	//Команды текущего шага
	(*1*) cmd_KR12_Off := drm.cmd.0 := TRUE; //Закрытие крана 12, открытие крана 9
	(*1*) drm.error.0 := am.KR12.notOff OR am.KR9.notOn; //Кран 12 не закрылся, кран 9 не открылся

	//Условие перехода (5)→(6)
	//Кран 12 закрылся И кран 9 открылся
	IF (am.KR12.isOFF AND am.KR9.isON) AND drm.timeout THEN
		drm.cmd := drm.error := 0; drm.timer_pt := cycle; drm.inc := FALSE; drm.step := 6;
		cmd_KR12_Off := FALSE; //Закрытие крана 12, открытие крана 9
	END_IF;
6:	//Запись уставки таймера шага
	drm.step := 6;//Текущий шаг
	drm.timer_pt := cycle; //Таймер: один цикл вызова

	//Команды текущего шага
	(*1*) cmd_Kr6_Off := drm.cmd.0 := TRUE; //Кран 6 закрыть
	(*1*) drm.error.0 := am.Kr6.notOff; //Кран 6 не закрылся

	//Условие перехода (6)→(7)
	//Кран 6 закрыт
	IF (am.Kr6.isOFF) AND drm.timeout THEN
		drm.cmd := drm.error := 0; drm.timer_pt := cycle; drm.inc := FALSE; drm.step := 7;
		cmd_Kr6_Off := FALSE; //Кран 6 закрыть
	END_IF;
7:	//Запись уставки таймера шага
	drm.step := 7;//Текущий шаг
	drm.timer_pt := cycle; //Таймер: один цикл вызова

	//Команды текущего шага
	(*1*) cmd_Kr1_Off := drm.cmd.0 := TRUE; //Кран 1 закрыть
	(*1*) drm.error.0 := am.Kr1.notOff; //Кран 1 не закрылся

	(*2*) cmd_Kr2_Off := drm.cmd.1 := TRUE; //Кран 2 закрыть
	(*2*) drm.error.1 := am.Kr2.notOff; //Кран 2 не закрылся

	(*3*) cmd_Kr4_On := drm.cmd.2 := TRUE; //Кран 4 открыть
	(*3*) drm.error.2 := am.Kr4.notOn; //Кран 4 не открылся

	//Условие перехода (7)→(8)
	//Кран 1 закрыт И Кран 2 закрыт И Кран 4 открыт
	IF (am.Kr1.isOFF AND am.Kr2.isOFF AND am.Kr4.isON) AND drm.timeout THEN
		drm.cmd := drm.error := 0; drm.timer_pt := cycle; drm.inc := FALSE; drm.step := 8;
		cmd_Kr1_Off := FALSE; //Кран 1 закрыть
		cmd_Kr2_Off := FALSE; //Кран 2 закрыть
		cmd_Kr4_On := FALSE; //Кран 4 открыть
	END_IF;
8:	//Запись уставки таймера шага
	drm.step := 8;//Текущий шаг
	drm.timer_pt := cycle; //Таймер: один цикл вызова

	//Команды текущего шага
	(*1*) finish := drm.cmd.0 := TRUE; //Завершение

	//Условие перехода (8)→(0)
	//Логическая 1
	IF (TRUE) AND drm.timeout THEN
		drm.cmd := drm.error := 0; drm.timer_pt := cycle; drm.inc := FALSE; drm.step := -1;
		finish := FALSE; //Завершение
	END_IF;
END_CASE

//Принудительный выход из последовательности
IF break THEN
	drm.step := -1; drm.cmd := drm.error := 0; drm.timer_pt := cycle; drm.inc := FALSE;
	cmd_sound_On := FALSE; //Предпусковая сигнализация
	cmd_PNU_S_On := FALSE; //Пуск маслонасосов уплотнения и смазки
	cmd_sh_dPmg_On := FALSE; //Взвод защиты по перепаду "масло-газ"
	cmd_shPmN_On := FALSE; //Взвод защиты по маслосистеме нагнетателя
	cmd_filling := FALSE; //Запуск последовательности "Заполнение контура компрессора"
	cmd_KR12_On := FALSE; //Открытие крана 12, закрытие крана 9
	cmd_KR12_Off := FALSE; //Закрытие крана 12, открытие крана 9
	cmd_Kr6_Off := FALSE; //Кран 6 закрыть
	cmd_Kr1_Off := FALSE; //Кран 1 закрыть
	cmd_Kr2_Off := FALSE; //Кран 2 закрыть
	cmd_Kr4_On := FALSE; //Кран 4 открыть
	finish := FALSE; //Завершение
END_IF;

                  
END_FUNCTION_BLOCK

{region INFO}
(*
 Наименование последовательности: Переход К-М
 Автор: /Разработчик/ 08.08.2025 9:04:03
 Версия: v00.00.18
 Проект: KA107
*)
{endregion}
{attribute 'symbol' := 'none'}
FUNCTION_BLOCK PUBLIC T_K_M
VAR_INPUT
	cycle : REAL; //цикл вызова
END_VAR
VAR_OUTPUT
	cmd_Kr2_On : BOOL; //Кран 2 открыть
	cmd_Kr6_Off : BOOL; //Кран 6 закрыть
	finish : BOOL; //Завершение
	{attribute 'symbol' := 'read'}
	drm : Tdrm; //Интерфейсный функциональный блок
END_VAR
VAR
	start : BOOL; //Запуск последовательности
	break : BOOL; //Принудительный выход из последовательности
END_VAR

                    //Собираем переходы для визуализации
drm.transition.0 := start := mde.K_M; //Запуск последовательности (0→1): (Режим Переход К-М)
drm.transition.1 := am.Kr2.isON; //1→2: Кран 2 открыт
drm.transition.2 := am.Kr6.isOff; //2→3: Кран 6 закрыт
drm.transition.3 := TRUE; //3→0: Логическая 1
drm.transition.31 := break := alg.AO OR mde.M_K; //Принудительный выход из последовательности (N→0): Режимы аварийного останова ИЛИ Режим "Переход М-К"

//Вызываем экземпляр интерфейсного функционального блока
drm(cycle := cycle);

CASE drm.step OF
-1:	//Сброс команд с предыдущих шагов
	finish := FALSE;
	//Условие запуска последовательности
	//(Режим Переход К-М)
	IF start AND NOT break THEN drm.step := 1; END_IF;
1:	//Запись уставки таймера шага
	drm.step := 1;//Текущий шаг
	drm.timer_pt := cycle; //Таймер: один цикл вызова

	//Команды текущего шага
	(*1*) cmd_Kr2_On := drm.cmd.0 := TRUE; //Кран 2 открыть
	(*1*) drm.error.0 := am.Kr2.notOn; //Кран 2 не открылся

	//Условие перехода (1)→(2)
	//Кран 2 открыт
	IF (am.Kr2.isON) AND drm.timeout THEN
		drm.cmd := drm.error := 0; drm.timer_pt := cycle; drm.inc := FALSE; drm.step := 2;
		cmd_Kr2_On := FALSE; //Кран 2 открыть
	END_IF;
2:	//Запись уставки таймера шага
	drm.step := 2;//Текущий шаг
	drm.timer_pt := cycle; //Таймер: один цикл вызова

	//Команды текущего шага
	(*1*) cmd_Kr6_Off := drm.cmd.0 := TRUE; //Кран 6 закрыть
	(*1*) drm.error.0 := am.Kr6.notOff; //Кран 6 не закрылся

	//Условие перехода (2)→(3)
	//Кран 6 закрыт
	IF (am.Kr6.isOff) AND drm.timeout THEN
		drm.cmd := drm.error := 0; drm.timer_pt := cycle; drm.inc := FALSE; drm.step := 3;
		cmd_Kr6_Off := FALSE; //Кран 6 закрыть
	END_IF;
3:	//Запись уставки таймера шага
	drm.step := 3;//Текущий шаг
	drm.timer_pt := cycle; //Таймер: один цикл вызова

	//Команды текущего шага
	(*1*) finish := drm.cmd.0 := TRUE; //Завершение

	//Условие перехода (3)→(0)
	//Логическая 1
	IF (TRUE) AND drm.timeout THEN
		drm.cmd := drm.error := 0; drm.timer_pt := cycle; drm.inc := FALSE; drm.step := -1;
		finish := FALSE; //Завершение
	END_IF;
END_CASE

//Принудительный выход из последовательности
IF break THEN
	drm.step := -1; drm.cmd := drm.error := 0; drm.timer_pt := cycle; drm.inc := FALSE;
	cmd_Kr2_On := FALSE; //Кран 2 открыть
	cmd_Kr6_Off := FALSE; //Кран 6 закрыть
	finish := FALSE; //Завершение
END_IF;

                  
END_FUNCTION_BLOCK

{region INFO}
(*
 Наименование последовательности: Переход М-К
 Автор: /Разработчик/ 08.08.2025 9:04:03
 Версия: v00.00.18
 Проект: KA107
*)
{endregion}
{attribute 'symbol' := 'none'}
FUNCTION_BLOCK PUBLIC T_M_K
VAR_INPUT
	cycle : REAL; //цикл вызова
END_VAR
VAR_OUTPUT
	cmd_KR6_On : BOOL; //Кран 6 открыть
	cmd_Kr2_Off : BOOL; //Кран 2 закрыть
	finish : BOOL; //Завершение
	{attribute 'symbol' := 'read'}
	drm : Tdrm; //Интерфейсный функциональный блок
END_VAR
VAR
	start : BOOL; //Запуск последовательности
	break : BOOL; //Принудительный выход из последовательности
END_VAR

                    //Собираем переходы для визуализации
drm.transition.0 := start := mde.M_K OR NOss.cmd_M_K OR NObs.cmd_M_K; //Запуск последовательности (0→1): (Режим Переход М-К) ИЛИ (НОсс => Переход М-К) ИЛИ (НОбс => Переход М-К)
drm.transition.1 := am.Kr6.isON; //1→2: Кран 6 открыт
drm.transition.2 := am.Kr2.isOFF; //2→3: Кран 2 закрыт
drm.transition.3 := TRUE; //3→0: Логическая 1
drm.transition.31 := break := mde.AOss OR mde.AObs OR mde.K_M; //Принудительный выход из последовательности (N→0): Режим АОсс ИЛИ Режим АОбс ИЛИ Режим "Переход К-М"

//Вызываем экземпляр интерфейсного функционального блока
drm(cycle := cycle);

CASE drm.step OF
-1:	//Сброс команд с предыдущих шагов
	finish := FALSE;
	//Условие запуска последовательности
	//(Режим Переход М-К) ИЛИ (НОсс => Переход М-К) ИЛИ (НОбс => Переход М-К)
	IF start AND NOT break THEN drm.step := 1; END_IF;
1:	//Запись уставки таймера шага
	drm.step := 1;//Текущий шаг
	drm.timer_pt := cycle; //Таймер: один цикл вызова

	//Команды текущего шага
	(*1*) cmd_KR6_On := drm.cmd.0 := TRUE; //Кран 6 открыть
	(*1*) drm.error.0 := am.KR6.notOn; //Кран 6 не открылся

	//Условие перехода (1)→(2)
	//Кран 6 открыт
	IF (am.Kr6.isON) AND drm.timeout THEN
		drm.cmd := drm.error := 0; drm.timer_pt := cycle; drm.inc := FALSE; drm.step := 2;
		cmd_KR6_On := FALSE; //Кран 6 открыть
	END_IF;
2:	//Запись уставки таймера шага
	drm.step := 2;//Текущий шаг
	drm.timer_pt := cycle; //Таймер: один цикл вызова

	//Команды текущего шага
	(*1*) cmd_Kr2_Off := drm.cmd.0 := TRUE; //Кран 2 закрыть
	(*1*) drm.error.0 := am.Kr2.notOff; //Кран 2 не закрылся

	//Условие перехода (2)→(3)
	//Кран 2 закрыт
	IF (am.Kr2.isOFF) AND drm.timeout THEN
		drm.cmd := drm.error := 0; drm.timer_pt := cycle; drm.inc := FALSE; drm.step := 3;
		cmd_Kr2_Off := FALSE; //Кран 2 закрыть
	END_IF;
3:	//Запись уставки таймера шага
	drm.step := 3;//Текущий шаг
	drm.timer_pt := cycle; //Таймер: один цикл вызова

	//Команды текущего шага
	(*1*) finish := drm.cmd.0 := TRUE; //Завершение

	//Условие перехода (3)→(0)
	//Логическая 1
	IF (TRUE) AND drm.timeout THEN
		drm.cmd := drm.error := 0; drm.timer_pt := cycle; drm.inc := FALSE; drm.step := -1;
		finish := FALSE; //Завершение
	END_IF;
END_CASE

//Принудительный выход из последовательности
IF break THEN
	drm.step := -1; drm.cmd := drm.error := 0; drm.timer_pt := cycle; drm.inc := FALSE;
	cmd_KR6_On := FALSE; //Кран 6 открыть
	cmd_Kr2_Off := FALSE; //Кран 2 закрыть
	finish := FALSE; //Завершение
END_IF;

                  
END_FUNCTION_BLOCK

{region INFO}
(*
 Наименование последовательности: НОбс
 Автор: /Разработчик/ 08.08.2025 9:04:03
 Версия: v00.00.18
 Проект: KA107
*)
{endregion}
{attribute 'symbol' := 'none'}
FUNCTION_BLOCK PUBLIC T_NObs
VAR_INPUT
	cycle : REAL; //цикл вызова
END_VAR
VAR_OUTPUT
	cmd_M_K : BOOL; //Запуск последовательности "Переход М-К"
	sh_ms_off : BOOL; //Снятие защиты по маслосистеме ТК и СТ
	cooling : BOOL; //Охлаждение двигателя
	cmd_PNU_S_On : BOOL; //Включение маслонасосов смазки и уплотнения
	cmd_VNA_On : BOOL; //Включение Э/М ВНА
	cmd_KPV234_On : BOOL; //Открыть КПВ 2, 3, 4
	cmd_KR12_Off : BOOL; //Закрытие крана 12, открытие крана 9
	cmd_sh_TG_Off : BOOL; //Снятие защиты по ТГ
	cmd_SK_Off : BOOL; //СК закрыть
	check_Nst : BOOL; //Выбег нагнетателя
	cmd_Kr1_Off : BOOL; //Кран 1 закрыть
	cmd_Kr6_Off : BOOL; //Кран 6 закрыть
	cmd_Kr4_On : BOOL; //Кран 4 открыть
	check_Ntk : BOOL; //Выбег двигателя
	finish : BOOL; //Завершение
	{attribute 'symbol' := 'read'}
	drm : Tdrm; //Интерфейсный функциональный блок
END_VAR
VAR
	start : BOOL; //Запуск последовательности
	break : BOOL; //Принудительный выход из последовательности
END_VAR

                    //Собираем переходы для визуализации
drm.transition.0 := start := mde.NObs; //Запуск последовательности (0→1): Режим НОбс
drm.transition.1 := M_K.finish; //1→2: Последовательность "Переход М-К" завершена
drm.transition.2 := FuelReg.fReg.cooling; //2→3: Двигатель перешел на малый газ для охлаждения
drm.transition.3 := NOT FuelReg.fReg.cooling; //3→4: Охлаждение двигателя завершено
drm.transition.4 := am.KR9.ison AND am.KR12.isOff; //4→5: Подача топливного газа прекращена
drm.transition.5 := acpar.Nst.value < 100.0; //5→6: Nст < 100 об/мин
drm.transition.6 := am.Kr1.isOFF AND am.Kr6.isOFF AND am.Kr4.isON; //6→7: Кран 1 закрыт И Кран 6 закрыт И Кран 4 открыт
drm.transition.7 := acpar.Ntk.value < 100.0; //7→8: Nтк < 100 об/мин
drm.transition.8 := TRUE; //8→0: Логическая 1
drm.transition.31 := break := mde.AObs; //Принудительный выход из последовательности (N→0): Режим АОбс

//Вызываем экземпляр интерфейсного функционального блока
drm(cycle := cycle);

CASE drm.step OF
-1:	//Сброс команд с предыдущих шагов
	finish := FALSE;
	//Условие запуска последовательности
	//Режим НОбс
	IF start AND NOT break THEN drm.step := 1; END_IF;
1:	//Запись уставки таймера шага
	drm.step := 1;//Текущий шаг
	drm.timer_pt := cycle; //Таймер: один цикл вызова

	//Команды текущего шага
	(*1*) cmd_M_K := drm.cmd.0 := drm.step_time <= cycle; //Запуск последовательности "Переход М-К"

	//Условие перехода (1)→(2)
	//Последовательность "Переход М-К" завершена
	IF (M_K.finish) AND drm.timeout THEN
		drm.cmd := drm.error := 0; drm.timer_pt := cycle; drm.inc := FALSE; drm.step := 2;
		cmd_M_K := FALSE; //Запуск последовательности "Переход М-К"
	END_IF;
2:	//Запись уставки таймера шага
	drm.step := 2;//Текущий шаг
	drm.timer_pt := 10; //Таймер: 10 секунд

	//Команды текущего шага
	(*1*) sh_ms_off := drm.cmd.0 := TRUE; //Снятие защиты по маслосистеме ТК и СТ

	(*2*) alg.normalStopCom := drm.cmd.1 := TRUE; //Нормальный останов двигателя
	(*2*) drm.error.1 := NOT FuelReg.fReg.cooling; //Д не перешел на малый газ для охлаждения

	//Условие перехода (2)→(3)
	//Двигатель перешел на малый газ для охлаждения
	IF (FuelReg.fReg.cooling) AND drm.timeout THEN
		drm.cmd := drm.error := 0; drm.timer_pt := cycle; drm.inc := FALSE; drm.step := 3;
		sh_ms_off := FALSE; //Снятие защиты по маслосистеме ТК и СТ
	END_IF;
3:	//Запись уставки таймера шага
	drm.step := 3;//Текущий шаг
	drm.inc := TRUE; //Выставляем признак инкремента

	//Команды текущего шага
	(*1*) cooling := drm.cmd.0 := TRUE; //Охлаждение двигателя

	//Условие перехода (3)→(4)
	//Охлаждение двигателя завершено
	IF (NOT FuelReg.fReg.cooling) AND drm.timeout THEN
		drm.cmd := drm.error := 0; drm.timer_pt := cycle; drm.inc := FALSE; drm.step := 4;
		cooling := FALSE; //Охлаждение двигателя
	END_IF;
4:	//Запись уставки таймера шага
	drm.step := 4;//Текущий шаг
	drm.timer_pt := cycle; //Таймер: один цикл вызова

	//Команды текущего шага
	(*1*) alg.normalStopCom := FALSE; //Нормальный останов двигателя

	(*2*) cmd_PNU_S_On := drm.cmd.1 := TRUE; //Включение маслонасосов смазки и уплотнения

	(*3*) cmd_VNA_On := drm.cmd.2 := TRUE; //Включение Э/М ВНА

	(*4*) cmd_KPV234_On := drm.cmd.3 := TRUE; //Открыть КПВ 2, 3, 4
	(*4*) drm.error.3 := am.KPV2.notOn OR am.KPV3.notOn OR am.KPV4.notOn; //КПВ 2, 3, 4 не открылись

	(*5*) cmd_KR12_Off := drm.cmd.4 := TRUE; //Закрытие крана 12, открытие крана 9
	(*5*) drm.error.4 := am.KR12.notOff OR am.KR9.notOn; //Кран 12 не закрылся, кран 9 не открылся

	(*6*) cmd_sh_TG_Off := drm.cmd.5 := TRUE; //Снятие защиты по ТГ

	(*7*) cmd_SK_Off := drm.cmd.6 := TRUE; //СК закрыть

	//Условие перехода (4)→(5)
	//Подача топливного газа прекращена
	IF (am.KR9.ison AND am.KR12.isOff) AND drm.timeout THEN
		drm.cmd := drm.error := 0; drm.timer_pt := cycle; drm.inc := FALSE; drm.step := 5;
		cmd_PNU_S_On := FALSE; //Включение маслонасосов смазки и уплотнения
		cmd_KPV234_On := FALSE; //Открыть КПВ 2, 3, 4
		cmd_KR12_Off := FALSE; //Закрытие крана 12, открытие крана 9
		cmd_sh_TG_Off := FALSE; //Снятие защиты по ТГ
		cmd_SK_Off := FALSE; //СК закрыть
	END_IF;
5:	//Запись уставки таймера шага
	drm.step := 5;//Текущий шаг
	drm.timer_pt := cycle; //Таймер: один цикл вызова

	//Команды текущего шага
	(*1*) check_Nst := drm.cmd.0 := TRUE; //Выбег нагнетателя

	//Условие перехода (5)→(6)
	//Nст < 100 об/мин
	IF (acpar.Nst.value < 100.0) AND drm.timeout THEN
		drm.cmd := drm.error := 0; drm.timer_pt := cycle; drm.inc := FALSE; drm.step := 6;
		check_Nst := FALSE; //Выбег нагнетателя
	END_IF;
6:	//Запись уставки таймера шага
	drm.step := 6;//Текущий шаг
	drm.timer_pt := cycle; //Таймер: один цикл вызова

	//Команды текущего шага
	(*1*) cmd_Kr1_Off := drm.cmd.0 := TRUE; //Кран 1 закрыть
	(*1*) drm.error.0 := am.Kr1.notOff; //Кран 1 не закрылся

	(*2*) cmd_Kr6_Off := drm.cmd.1 := TRUE; //Кран 6 закрыть
	(*2*) drm.error.1 := am.Kr6.notOff; //Кран 6 не закрылся

	(*3*) cmd_Kr4_On := drm.cmd.2 := TRUE; //Кран 4 открыть
	(*3*) drm.error.2 := am.Kr4.notOn; //Кран 4 не открылся

	//Условие перехода (6)→(7)
	//Кран 1 закрыт И Кран 6 закрыт И Кран 4 открыт
	IF (am.Kr1.isOFF AND am.Kr6.isOFF AND am.Kr4.isON) AND drm.timeout THEN
		drm.cmd := drm.error := 0; drm.timer_pt := cycle; drm.inc := FALSE; drm.step := 7;
		cmd_Kr1_Off := FALSE; //Кран 1 закрыть
		cmd_Kr6_Off := FALSE; //Кран 6 закрыть
		cmd_Kr4_On := FALSE; //Кран 4 открыть
	END_IF;
7:	//Запись уставки таймера шага
	drm.step := 7;//Текущий шаг
	drm.timer_pt := cycle; //Таймер: один цикл вызова

	//Команды текущего шага
	(*1*) check_Ntk := drm.cmd.0 := TRUE; //Выбег двигателя

	//Условие перехода (7)→(8)
	//Nтк < 100 об/мин
	IF (acpar.Ntk.value < 100.0) AND drm.timeout THEN
		drm.cmd := drm.error := 0; drm.timer_pt := cycle; drm.inc := FALSE; drm.step := 8;
		check_Ntk := FALSE; //Выбег двигателя
	END_IF;
8:	//Запись уставки таймера шага
	drm.step := 8;//Текущий шаг
	drm.timer_pt := cycle; //Таймер: один цикл вызова

	//Команды текущего шага
	(*1*) cmd_VNA_On := FALSE; //Отключение Э/М ВНА

	(*2*) finish := drm.cmd.1 := drm.step_time <= cycle; //Завершение

	//Условие перехода (8)→(0)
	//Логическая 1
	IF (TRUE) AND drm.timeout THEN
		drm.cmd := drm.error := 0; drm.timer_pt := cycle; drm.inc := FALSE; drm.step := -1;
		finish := FALSE; //Завершение
	END_IF;
END_CASE

//Принудительный выход из последовательности
IF break THEN
	drm.step := -1; drm.cmd := drm.error := 0; drm.timer_pt := cycle; drm.inc := FALSE;
	cmd_M_K := FALSE; //Запуск последовательности "Переход М-К"
	sh_ms_off := FALSE; //Снятие защиты по маслосистеме ТК и СТ
	alg.normalStopCom := FALSE; //Нормальный останов двигателя
	cooling := FALSE; //Охлаждение двигателя
	cmd_PNU_S_On := FALSE; //Включение маслонасосов смазки и уплотнения
	cmd_VNA_On := FALSE; //Включение Э/М ВНА
	cmd_KPV234_On := FALSE; //Открыть КПВ 2, 3, 4
	cmd_KR12_Off := FALSE; //Закрытие крана 12, открытие крана 9
	cmd_sh_TG_Off := FALSE; //Снятие защиты по ТГ
	cmd_SK_Off := FALSE; //СК закрыть
	check_Nst := FALSE; //Выбег нагнетателя
	cmd_Kr1_Off := FALSE; //Кран 1 закрыть
	cmd_Kr6_Off := FALSE; //Кран 6 закрыть
	cmd_Kr4_On := FALSE; //Кран 4 открыть
	check_Ntk := FALSE; //Выбег двигателя
	finish := FALSE; //Завершение
END_IF;

                  
END_FUNCTION_BLOCK

{region INFO}
(*
 Наименование последовательности: НОсс
 Автор: /Разработчик/ 08.08.2025 9:04:03
 Версия: v00.00.18
 Проект: KA107
*)
{endregion}
{attribute 'symbol' := 'none'}
FUNCTION_BLOCK PUBLIC T_NOss
VAR_INPUT
	cycle : REAL; //цикл вызова
END_VAR
VAR_OUTPUT
	cmd_M_K : BOOL; //Запуск последовательности "Переход М-К"
	sh_ms_off : BOOL; //Снятие защиты по маслосистеме ТК и СТ
	cooling : BOOL; //Охлаждение двигателя
	cmd_PNU_S_On : BOOL; //Включение маслонасосов смазки и уплотнения
	cmd_VNA_On : BOOL; //Включение Э/М ВНА
	cmd_KPV234_On : BOOL; //Открыть КПВ 2, 3, 4
	cmd_KR12_Off : BOOL; //Закрытие крана 12, открытие крана 9
	cmd_sh_TG_Off : BOOL; //Снятие защиты по ТГ
	cmd_SK_Off : BOOL; //СК закрыть
	check_Nst : BOOL; //Выбег нагнетателя
	cmd_bleeding : BOOL; //Запуск последовательности "Стравливание контура компрессора"
	cmd_sh_dPmg_Off : BOOL; //Снятие защиты по перепаду "масло-газ"
	cmd_PNU_S_Off : BOOL; //Пуск таймера отключения ПНС, ПНУ
	check_Ntk : BOOL; //Выбег двигателя
	cmd_shPmN_Off : BOOL; //Снятие защиты по маслосистеме нагнетателя
	finish : BOOL; //Завершение
	{attribute 'symbol' := 'read'}
	drm : Tdrm; //Интерфейсный функциональный блок
END_VAR
VAR
	start : BOOL; //Запуск последовательности
	break : BOOL; //Принудительный выход из последовательности
END_VAR

                    //Собираем переходы для визуализации
drm.transition.0 := start := mde.NOss; //Запуск последовательности (0→1): Режим НОсс
drm.transition.1 := M_K.finish; //1→2: Последовательность "Переход М-К" завершена
drm.transition.2 := FuelReg.fReg.cooling; //2→3: Двигатель перешел на малый газ для охлаждения
drm.transition.3 := NOT FuelReg.fReg.cooling; //3→4: Охлаждение двигателя завершено
drm.transition.4 := am.KR9.ison AND am.KR12.isOff; //4→5: Подача топливного газа прекращена
drm.transition.5 := acpar.Nst.value < 100.0; //5→6: Nст < 100 об/мин
drm.transition.6 := bleeding.finish; //6→7: Подрежим "Стравливание контура компрессора" завершен
drm.transition.7 := acpar.Ntk.value < 100.0; //7→8: Nтк < 100 об/мин
drm.transition.8 := TRUE; //8→0: Логическая 1
drm.transition.31 := break := mde.AOss; //Принудительный выход из последовательности (N→0): Режим АОсс

//Вызываем экземпляр интерфейсного функционального блока
drm(cycle := cycle);

CASE drm.step OF
-1:	//Сброс команд с предыдущих шагов
	finish := FALSE;
	//Условие запуска последовательности
	//Режим НОсс
	IF start AND NOT break THEN drm.step := 1; END_IF;
1:	//Запись уставки таймера шага
	drm.step := 1;//Текущий шаг
	drm.timer_pt := cycle; //Таймер: один цикл вызова

	//Команды текущего шага
	(*1*) cmd_M_K := drm.cmd.0 := drm.step_time <= cycle; //Запуск последовательности "Переход М-К"

	//Условие перехода (1)→(2)
	//Последовательность "Переход М-К" завершена
	IF (M_K.finish) AND drm.timeout THEN
		drm.cmd := drm.error := 0; drm.timer_pt := cycle; drm.inc := FALSE; drm.step := 2;
		cmd_M_K := FALSE; //Запуск последовательности "Переход М-К"
	END_IF;
2:	//Запись уставки таймера шага
	drm.step := 2;//Текущий шаг
	drm.timer_pt := 10; //Таймер: 10 секунд

	//Команды текущего шага
	(*1*) sh_ms_off := drm.cmd.0 := TRUE; //Снятие защиты по маслосистеме ТК и СТ

	(*2*) alg.normalStopCom := drm.cmd.1 := TRUE; //Нормальный останов двигателя
	(*2*) drm.error.1 := NOT FuelReg.fReg.cooling; //Д не перешел на малый газ для охлаждения

	//Условие перехода (2)→(3)
	//Двигатель перешел на малый газ для охлаждения
	IF (FuelReg.fReg.cooling) AND drm.timeout THEN
		drm.cmd := drm.error := 0; drm.timer_pt := cycle; drm.inc := FALSE; drm.step := 3;
		sh_ms_off := FALSE; //Снятие защиты по маслосистеме ТК и СТ
	END_IF;
3:	//Запись уставки таймера шага
	drm.step := 3;//Текущий шаг
	drm.inc := TRUE; //Выставляем признак инкремента

	//Команды текущего шага
	(*1*) cooling := drm.cmd.0 := TRUE; //Охлаждение двигателя

	//Условие перехода (3)→(4)
	//Охлаждение двигателя завершено
	IF (NOT FuelReg.fReg.cooling) AND drm.timeout THEN
		drm.cmd := drm.error := 0; drm.timer_pt := cycle; drm.inc := FALSE; drm.step := 4;
		cooling := FALSE; //Охлаждение двигателя
	END_IF;
4:	//Запись уставки таймера шага
	drm.step := 4;//Текущий шаг
	drm.timer_pt := cycle; //Таймер: один цикл вызова

	//Команды текущего шага
	(*1*) alg.normalStopCom := FALSE; //Нормальный останов двигателя

	(*2*) cmd_PNU_S_On := drm.cmd.1 := TRUE; //Включение маслонасосов смазки и уплотнения

	(*3*) cmd_VNA_On := drm.cmd.2 := TRUE; //Включение Э/М ВНА

	(*4*) cmd_KPV234_On := drm.cmd.3 := TRUE; //Открыть КПВ 2, 3, 4
	(*4*) drm.error.3 := am.KPV2.notOn OR am.KPV3.notOn OR am.KPV4.notOn; //КПВ 2, 3, 4 не открылись

	(*5*) cmd_KR12_Off := drm.cmd.4 := TRUE; //Закрытие крана 12, открытие крана 9
	(*5*) drm.error.4 := am.KR12.notOff OR am.KR9.notOn; //Кран 12 не закрылся, кран 9 не открылся

	(*6*) cmd_sh_TG_Off := drm.cmd.5 := TRUE; //Снятие защиты по ТГ

	(*7*) cmd_SK_Off := drm.cmd.6 := TRUE; //СК закрыть

	//Условие перехода (4)→(5)
	//Подача топливного газа прекращена
	IF (am.KR9.ison AND am.KR12.isOff) AND drm.timeout THEN
		drm.cmd := drm.error := 0; drm.timer_pt := cycle; drm.inc := FALSE; drm.step := 5;
		cmd_PNU_S_On := FALSE; //Включение маслонасосов смазки и уплотнения
		cmd_KPV234_On := FALSE; //Открыть КПВ 2, 3, 4
		cmd_KR12_Off := FALSE; //Закрытие крана 12, открытие крана 9
		cmd_sh_TG_Off := FALSE; //Снятие защиты по ТГ
		cmd_SK_Off := FALSE; //СК закрыть
	END_IF;
5:	//Запись уставки таймера шага
	drm.step := 5;//Текущий шаг
	drm.timer_pt := cycle; //Таймер: один цикл вызова

	//Команды текущего шага
	(*1*) check_Nst := drm.cmd.0 := TRUE; //Выбег нагнетателя

	//Условие перехода (5)→(6)
	//Nст < 100 об/мин
	IF (acpar.Nst.value < 100.0) AND drm.timeout THEN
		drm.cmd := drm.error := 0; drm.timer_pt := cycle; drm.inc := FALSE; drm.step := 6;
		check_Nst := FALSE; //Выбег нагнетателя
	END_IF;
6:	//Запись уставки таймера шага
	drm.step := 6;//Текущий шаг
	drm.timer_pt := cycle; //Таймер: один цикл вызова

	//Команды текущего шага
	(*1*) cmd_bleeding := drm.cmd.0 := drm.step_time <= cycle; //Запуск последовательности "Стравливание контура компрессора"

	//Условие перехода (6)→(7)
	//Подрежим "Стравливание контура компрессора" завершен
	IF (bleeding.finish) AND drm.timeout THEN
		drm.cmd := drm.error := 0; drm.timer_pt := cycle; drm.inc := FALSE; drm.step := 7;
		cmd_bleeding := FALSE; //Запуск последовательности "Стравливание контура компрессора"
	END_IF;
7:	//Запись уставки таймера шага
	drm.step := 7;//Текущий шаг
	drm.timer_pt := 2; //Таймер: 2 секунд

	//Команды текущего шага
	(*1*) cmd_sh_dPmg_Off := drm.cmd.0 := TRUE; //Снятие защиты по перепаду "масло-газ"

	(*2*) cmd_PNU_S_Off := drm.cmd.1 := drm.step_time <= cycle; //Пуск таймера отключения ПНС, ПНУ

	(*3*) check_Ntk := drm.cmd.2 := TRUE; //Выбег двигателя

	//Условие перехода (7)→(8)
	//Nтк < 100 об/мин
	IF (acpar.Ntk.value < 100.0) AND drm.timeout THEN
		drm.cmd := drm.error := 0; drm.timer_pt := cycle; drm.inc := FALSE; drm.step := 8;
		cmd_sh_dPmg_Off := FALSE; //Снятие защиты по перепаду "масло-газ"
		cmd_PNU_S_Off := FALSE; //Пуск таймера отключения ПНС, ПНУ
		check_Ntk := FALSE; //Выбег двигателя
	END_IF;
8:	//Запись уставки таймера шага
	drm.step := 8;//Текущий шаг
	drm.timer_pt := cycle; //Таймер: один цикл вызова

	//Команды текущего шага
	(*1*) cmd_VNA_On := FALSE; //Отключение Э/М ВНА

	(*2*) cmd_shPmN_Off := drm.cmd.1 := TRUE; //Снятие защиты по маслосистеме нагнетателя

	(*3*) cmd_PNU_S_Off := drm.cmd.2 := drm.step_time <= cycle; //Пуск таймера отключения ПНС, ПНУ

	(*4*) finish := drm.cmd.3 := TRUE; //Завершение

	//Условие перехода (8)→(0)
	//Логическая 1
	IF (TRUE) AND drm.timeout THEN
		drm.cmd := drm.error := 0; drm.timer_pt := cycle; drm.inc := FALSE; drm.step := -1;
		cmd_shPmN_Off := FALSE; //Снятие защиты по маслосистеме нагнетателя
		cmd_PNU_S_Off := FALSE; //Пуск таймера отключения ПНС, ПНУ
		finish := FALSE; //Завершение
	END_IF;
END_CASE

//Принудительный выход из последовательности
IF break THEN
	drm.step := -1; drm.cmd := drm.error := 0; drm.timer_pt := cycle; drm.inc := FALSE;
	cmd_M_K := FALSE; //Запуск последовательности "Переход М-К"
	sh_ms_off := FALSE; //Снятие защиты по маслосистеме ТК и СТ
	alg.normalStopCom := FALSE; //Нормальный останов двигателя
	cooling := FALSE; //Охлаждение двигателя
	cmd_PNU_S_On := FALSE; //Включение маслонасосов смазки и уплотнения
	cmd_VNA_On := FALSE; //Включение Э/М ВНА
	cmd_KPV234_On := FALSE; //Открыть КПВ 2, 3, 4
	cmd_KR12_Off := FALSE; //Закрытие крана 12, открытие крана 9
	cmd_sh_TG_Off := FALSE; //Снятие защиты по ТГ
	cmd_SK_Off := FALSE; //СК закрыть
	check_Nst := FALSE; //Выбег нагнетателя
	cmd_bleeding := FALSE; //Запуск последовательности "Стравливание контура компрессора"
	cmd_sh_dPmg_Off := FALSE; //Снятие защиты по перепаду "масло-газ"
	cmd_PNU_S_Off := FALSE; //Пуск таймера отключения ПНС, ПНУ
	check_Ntk := FALSE; //Выбег двигателя
	cmd_shPmN_Off := FALSE; //Снятие защиты по маслосистеме нагнетателя
	cmd_PNU_S_Off := FALSE; //Пуск таймера отключения ПНС, ПНУ
	finish := FALSE; //Завершение
END_IF;

                  
END_FUNCTION_BLOCK

///
/// Назначение: 		Подготовка данных и вызхов обработчиков сигнализаций
/// Версия: 			00.00.00
/// Проект: 			КА107
FUNCTION Alarm_link : BOOL

                    //Деблокировка
unlock := tch.Unlock.value := btn.Unlock.out;

//Проверка защит
tch.CheckAlarm_on.value := btn.CheckAlarm_on.out OR tch.CheckAlarm_on.value AND NOT btn.CheckAlarm_off.out;
crs.common.CheckAlarm := alr.common.CheckAlarm := tch.CheckAlarm_on.value; 

// Подготовка данных для обработчиков сигнализаций	 
// Включение защиты по маслосистеме воздушного стартера
tmr.crsPmStarter_20.in 	:= am.Kr13.on;
alg.sh_Starter 			:= tmr.crsPmStarter_20.q;

// Защита по топливному газу
alg.sh_TG	:= ( Start_D.cmd_sh_TG_On OR alg.sh_TG ) AND NOT ( NOss.cmd_sh_TG_Off OR NObs.cmd_sh_TG_Off OR AOss.cmd_sh_TG_Off OR AObs.cmd_sh_TG_Off ) OR tch.GTDwork.value;

// Включение защиты по не розжигу (10 sec)
//tmr.crsNIgnition_10.IN	:= Start_D.cmd_sh_nIgnition AND NOT FuelReg.fReg.isFire;
alg.sh_nIgnition 		:= Start_D.cmd_sh_nIgnition AND NOT FuelReg.fReg.isFire; //tmr.crsNIgnition_10.Q;

// Включение защиты по не раскрутке (10 sec)
//tmr.crsNBoost_10.IN		:= ( Start_D.cmd_sh_nBoost OR tmr.crsNBoost_10.IN ) AND acpar.Ntk.value < 5600 AND am.SK.on;
alg.sh_nBoost			:= ( Start_D.cmd_sh_nBoost ) AND acpar.Ntk.value < 5600 AND am.SK.on; //tmr.crsNBoost_10.Q;

// Взвод защиты КПВ234 не закрыты
tmr.KPV234_wOpen.IN		:= ( Start_D.cmd_KPV234_Off OR tmr.KPV234_wOpen.IN ) AND NOT tmr.KPV234_wOpen.Q;
alg.KPV234_wOpen		:= ( tmr.KPV234_wOpen.Q OR alg.KPV234_wOpen ) AND NOT ( NOss.cmd_KPV234_On OR NObs.cmd_KPV234_On OR AOss.cmd_KPV234_On OR AObs.cmd_KPV234_On ) OR tch.GTDwork.value;

// Взвод защиты КПВ15 не закрыты
tmr.KPV15_wOpen.IN		:= ( acpar.NtkPrived.value > Ntk_KPV15Close OR tmr.KPV15_wOpen.IN ) AND NOT ( AOss.cmd_KPV15_On OR AObs.cmd_KPV15_On OR alg.normalStopCom );
alg.KPV15_wOpen			:= tmr.KPV15_wOpen.Q;

// Взвод защиты КПВ15 не открыты
tmr.KPV15_nOpen.IN		:= ( acpar.NtkPrived.value < Ntk_KPV15Open ) AND ( acpar.NtkPrived.value > Ntk_KPVClose );
alg.KPV15_nOpen			:= tmr.KPV15_nOpen.Q;

// Взвод защиты по давлению газа перед краном 13
alg.sh_Pg_inKR13		:= ( HP.cmd_VS_On OR Start_D.cmd_VS_On OR alg.sh_Pg_inKR13 ) AND NOT ( HP.cmd_VS_Off OR Start_D.cmd_VS_Off );

// Взвод защиты по давлению масла нагнетателя
alg.sh_PmN				:= ( KPK.cmd_shPmN_On OR HP.cmd_shPmN_On OR APK.cmd_shPmN_On OR alg.sh_PmN ) AND NOT ( HP.cmd_shPmN_Off OR NOss.cmd_shPmN_Off OR AOss.cmd_shPmN_Off OR Bleeding_full.cmd_shPmN_Off ) OR tch.GTDwork.value;

// Взвод защиты по давлению масла ТК и СТ
alg.sh_PmGTD			:= alg.KPV15_wOpen;

// Взвод защиты по давлению масла перед ДГ (САР)
alg.sh_SAR				:= alg.KPV234_wOpen;

// Взвод защиты по перепаду масло-газ
alg.sh_dPmg				:= ( KPK.cmd_sh_dPmg_On OR HP.cmd_sh_dPmg_On OR APK.cmd_sh_dPmg_On OR alg.sh_dPmg ) AND NOT ( HP.cmd_sh_dPmg_Off OR NOss.cmd_sh_dPmg_Off OR AOss.cmd_sh_dPmg_Off OR Bleeding_full.cmd_sh_dPmg_Off ) OR tch.Gas_N.value;

// Аварийный останов
alg.emergStopCom		:= AOss.emergStopCom OR AObs.emergStopCom;

// Вызов обработчиков сигнализаций
PPU_update(); // Предпусковые условия
ALR_update(); // Предупреждения
CRS_update(); // Аварии
                  
END_FUNCTION

FUNCTION ALG_D_link : BOOL

                    
subsystem.BD(
	goWork := FuelReg.fReg.start OR HP.cmd_HP_D,
	work := tch.GTDwork.value OR mde.HP AND acpar.Ntk.value > 500.0, 
	stop := acpar.Ntk.value < 100.0);
	
//Автоформируемый вызов последовательностей
bd_update(cycle := cycle_time_base);

ALG_D_AM_base();

// Сигнал "ГТД в работе"
tch.GTDwork.value 	:= FuelReg.fReg.started;
// Сигнал "Прогрев ГТД"
tch.GTDHeat.value	:= FuelReg.fReg.heating;
// Сигнал "Охлаждение двигателя"
tch.GTDcool.value	:= FuelReg.fReg.cooling;
// Сигнал "Пуск агрегата"
tch.GTDstart.value	:= FuelReg.fReg.start;

//engine.work8h(IN := tch.GTDwork.value);
//engine.work12h(IN := tch.GTDwork.value);

IF imitGPA.imit_on THEN D_imit(); END_IF;
                  
END_FUNCTION

///Chekmarev
FUNCTION D_imit : BOOL
VAR
	Tm		: REAL; //  
	///start		: BOOL;
	PmGood	: BOOL;
END_VAR
VAR CONSTANT
	/// максимальные обороты ТК на стартере
	Nstart_max: REAL := 2050;
	/// номинальные обороты ТК
	Ntk_norm: REAL := 8300;
	// нагрев масла нагревателем
	Ten		: REAL := 65;
	/// нагрев масла двигателем
	dTm_max: REAL := 26;
	tau_m: REAL := (300 * cycle_time_base);
	tau_mb: REAL := (5000 * cycle_time_base);
END_VAR

                    //start := am.Kr11.isON AND am.Kr10.isOFF AND am.Kr13.on;

// Раскрутка стартером
//IF am.SK.isOFF AND start THEN
//	aipar.Ntk_1.sim_value := aipar.Ntk_1.value + ( Nstart_max - aipar.Ntk_1.value ) / tau_start;
//END_IF

// Выбег двигателя
//IF am.SK.isOFF AND NOT start THEN
//	aipar.Ntk_1.sim_value := aipar.Ntk_1.value - aipar.Ntk_1.value / tau_stop;
//END_IF

//aipar.Ntk_2.sim_value := aipar.Ntk_1.value + ( 10 * BOOL_TO_BYTE (aipar.Ntk_1.value > 10.0 ));

// Температура масла
Tm	:= aipar.Tm_outAVOM.value;
aipar.Tm_MB.sim_value	:= aipar.Tm_MB.value + ( Tm - aipar.Tm_MB.value) / tau_mb;	// в маслобаке
aipar.Tm_outD.sim_value	:= aipar.Tm_outD.sim_value + (aipar.Tm_inD.value + dTm_max * ( acpar.Ntk.value / Ntk_norm) - aipar.Tm_outD.sim_value) / tau_m;
aipar.Tm_inD.sim_value	:= aipar.Tm_MB.value - 0.5;		// на входе в двигатель
Tm	:= aipar.Tm_outAVOM.value;
aipar.Tm_MBU.sim_value	:= aipar.Tm_MBU.value + ( Tm - aipar.Tm_MBU.value ) / ( tau_mb * 5 ); // маслобак уплотнений

// q = 160 кг в мин // расход
// Q = 8380000 дж в мин // передача теплоты в масло
// ~ 2000 дж/(кгС) // теплоемкость масла
// Итог:
// dt = ~26 градусов за мин

PmGood	:= acpar.Ntk.value > 5000;

dipar.Pm_N_An.sim_value	:= NOT ( am.PNS.isOn OR PmGood );
dipar.Pm_N_Pn.sim_value := NOT ( am.PNS.isOn OR acpar.Ntk.value > 6880 );
dipar.Pm_TK_An.sim_value := acpar.Ntk.value < 7700;
dipar.Pm_ST_An.sim_value := dipar.Pm_TK_An.value;

// БЗА Готовность 2
dipar.BZA_ready_2.sim_value	:= PmGood;

// Положение концевиков КПВ
dipar.KPV1_ON.sim_value	:= acpar.Ntk.value > Ntk_KPVClose AND acpar.Ntk.value < 7710;
dipar.KPV1_off.sim_value	:= NOT ( acpar.Ntk.value > Ntk_KPVClose AND acpar.Ntk.value < 7500 );

dipar.KPV2_ON.sim_value	:= am.KPV2.ON AND PmGood;
dipar.KPV2_off.sim_value	:= NOT dipar.KPV2_ON.value;

dipar.KPV3_ON.sim_value	:= am.KPV3.ON AND PmGood;
dipar.KPV3_off.sim_value	:= NOT dipar.KPV3_ON.value;

dipar.KPV4_ON.sim_value	:= am.KPV4.ON AND PmGood;
dipar.KPV4_off.sim_value	:= NOT dipar.KPV4_ON.value;

dipar.KPV5_ON.sim_value	:= dipar.KPV1_ON.value;
dipar.KPV5_off.sim_value	:= dipar.KPV1_off.value;
                  
END_FUNCTION

FUNCTION ALG_base : BOOL

                    //Предпусковые подрежимы
//Режимы
	ALG_Modes_link();

//Подсистемы
	ALG_EXT_Link();
	ALG_BTG_Link();
	ALG_MSD_link();
 	ALG_GO_link();
 	ALG_D_link();
 	ALG_BN_link();
	ALG_AVOM_Link();
	ALG_BPG_Link();
	ALG_VS_Link();
	ALG_VOU_Link();
	ALG_BU_Link();

//Подрежимы
	ALG_SMD_link();
	

	check_modes();	
//Общие ИМы
	ALG_AM();

//Имитация
	imit();

//Тестирование алгоритмов
//	test_function();
                  
END_FUNCTION

FUNCTION ALG_Modes_link : BOOL

                    //Вызов графа режимов	
mde_update();
mde_hmi.number := mde.number;
mde_hmi.status.0 := GVL_LIB.DU_prm_all;
mde_hmi.status.1 := GVL_LIB.sim_on_all;
mde_hmi.status.2 := alr.common.type_aggregated.1;
mde_hmi.status.3 := trs.common.type_aggregated.3 OR crs.common.aggregated;
mde_hmi.status.4 := lmt.common.type_aggregated.2 OR FuelReg.fReg.commonLimUp OR FuelReg.fReg.commonLimDn;
mde_hmi.status.5 := aipar.common.sim_aggregated OR aopar.common.sim_aggregated OR dipar.common.sim_aggregated OR dopar.common.sim_aggregated;
mde_hmi.status.6 := aipar.common.flt_aggregated;
mde_hmi.status.7 := aopar.common.flt_aggregated;
mde_hmi.status.8 := dipar.common.flt_aggregated;
mde_hmi.status.9 := dopar.common.flt_aggregated;

//Обобщенные сигналы
alg.stop := mde.AOss OR mde.AObs OR mde.NOss OR mde.NObs;
alg.reserve := mde.HR OR mde.GR;
alg.V_000 := alg.reserve OR mde.Repair;
alg.test := mde.HP OR mde.KPK;
alg.start := mde.APK;
alg.work := mde.K OR mde.M OR mde.K_M OR mde.M_K;
alg.AO := mde.AOss OR mde.AObs;
alg.NO := mde.NOss OR mde.NObs;
                  
END_FUNCTION

///
/// Назначение: 		Инициализация переменных
/// Автор: 			
/// Версия: 			00.00.01
FUNCTION fun_init : BOOL

                    
//Инициализация при запуске контроллера

btn.imit_ON.cmd := TRUE; //включение имитации

// Инициализация АВОМ
AVOM_Init();

// Запрет расчёта uccV на термопарах
aipar.Tg_inST_1.cfg.ucv_enabled := FALSE;
aipar.Tg_inST_2.cfg.ucv_enabled := FALSE;
aipar.Tg_inST_3.cfg.ucv_enabled := FALSE;
aipar.Tg_inST_4.cfg.ucv_enabled := FALSE;
aipar.Tg_inST_5.cfg.ucv_enabled := FALSE;
aipar.Tg_inST_6.cfg.ucv_enabled := FALSE;

// Инициализация FileManager
FilesNames.OperationTimePath := 'OpTime/';
FilesNames.OperationTimeFileExt := '.txt';
FilesNames.OperationTimeOut := 20000;	// Дпустимое время работы с файлами - 20 мс.
                  
END_FUNCTION

FUNCTION ALG_GO_AM : BOOL

                    
// Кран 1
am.Kr1.on 	:= Filling.cmd_Kr1_ON;
am.Kr1.off 	:= KPK.cmd_Kr1_Off OR NObs.cmd_Kr1_Off OR AObs.cmd_Kr1_Off OR Bleeding.cmd_Kr1_Off;
// Кран 1 смазка
dopar.Kr1m_ON.value	:= am.Kr1.offOut OR am.Kr1.onOut;

// Кран 2
//aspar.dP_Kr2.value := ABS(aipar.Pg_outN.value - aipar.Pg_aftKr2.value);
am.Kr2.on 	:= K_M.cmd_Kr2_ON;
am.Kr2.off	:= KPK.cmd_Kr2_Off OR M_K.cmd_Kr2_Off OR AObs.cmd_Kr2_Off OR Bleeding.cmd_Kr2_Off;
// Кран 2 смазка
dopar.Kr2m_ON.value	:= am.Kr2.offOut OR am.Kr2.onOut;

// Кран 4
am.Kr4.on 	:= Filling.cmd_Kr4_ON OR KPK.cmd_Kr4_ON OR NObs.cmd_Kr4_ON OR AObs.cmd_Kr4_ON;
am.Kr4.off 	:= Filling.cmd_Kr4_Off OR Bleeding.cmd_Kr4_Off OR AOss.cmd_Kr4_Off OR AObs.cmd_Kr4_Off;
// Кран 4 смазка
//dopar.Kr4m_ON.value	:= am.Kr4.offOut OR am.Kr4.onOut;

// Кран 5
am.Kr5.on 	:= Bleeding.cmd_Kr5_ON AND am.Kr6.isOFF;
am.Kr5.off 	:= Filling.cmd_Kr5_Off;
// Кран 5 смазка
//dopar.Kr5m_ON.value	:= am.Kr5.offOut OR am.Kr5.onOut;

// Кран 6
am.Kr6.on 	:= M_K.cmd_KR6_ON OR Filling.cmd_Kr6_ON OR s_tunpar.ASprot.emergOpenBypass;
am.Kr6.off 	:= K_M.cmd_Kr6_Off OR NObs.cmd_Kr6_Off OR Bleeding.cmd_Kr6_Off OR AObs.cmd_Kr6_Off OR KPK.cmd_Kr6_Off OR ( alg.KR6_off_after_emergOpenBypass.Qr AND mde.M );
// Кран 6 смазка
dopar.Kr6m_ON.value	:= am.Kr6.offOut OR am.Kr6.onOut;
                  
END_FUNCTION

///
/// Назначение: 		Управление крановой обвязкой
/// Автор: 			
/// Версия: 			00.00.01
FUNCTION ALG_GO_link : BOOL

                    
subsystem.GO(
	goWork := filling.start, 
	goStop := bleeding.start, 
	work := filling.finish, 
	stop := bleeding.finish);
//Автоформируемый вызов последовательностей
go_update(cycle := cycle_time_base);

//Исполнительные механизмы
ALG_GO_AM();

//Нет газа в контуре Компрессора
tch.nGas_N.value := aipar.Pg_inN.value < 0.05 AND aipar.Pg_outN.value < 0.05 AND dipar.Kr5_ON.value AND NOT dipar.Kr5_off.value;
//Газ в контуре Компрессора
tch.Gas_N.value := (aipar.Pg_inN.value > 0.2 OR aipar.Pg_outN.value > 0.2) AND dipar.Kr5_off.value AND NOT dipar.Kr5_ON.value OR aipar.Pg_inN.value > 0.2 AND aipar.Pg_outN.value > 0.2;

//Нет роста Рг на вх. К на 0,05 МПа в течении 10 сек
IF aipar.Pg_inN.value - Pg_inN_old < 0.05 THEN
	bn.delay_filling := bn.delay_filling + cycle_time_base;
	IF bn.delay_filling > 10.0 THEN bn.delay_filling := 0.0; alg.nIncPgN := TRUE; END_IF;
ELSE
	alg.nIncPgN := FALSE;
END_IF;
Pg_inN_old := aipar.Pg_inN.value;

// выделение заднего фронта (снятия) предпомпажной защиты
alg.KR6_off_after_emergOpenBypass.in := s_tunpar.ASprot.emergOpenBypass;

IF imitGPA.imit_on THEN GO_imit(); END_IF;
                  
END_FUNCTION

///Chekmarev
FUNCTION GO_imit : BOOL
VAR
	tau: REAL;
	p_in: REAL;
	kx: REAL;
END_VAR
VAR CONSTANT
	/// 30.6 кгс
	Pg_in: REAL := 3;
	Pg_out_max: REAL := 7;
	Nst_max: REAL := 8400;
END_VAR

                    
kx := (Pg_out_max - Pg_in) / Nst_max * BOOL_TO_INT( am.Kr6.isOFF );

//Давление газа в Н
IF NOT dipar.Kr5_off.value THEN 
	tau := 20.0; 
ELSIF dipar.Kr4_ON.value THEN 
	tau := 50.0; 
ELSIF (dipar.Kr1_ON.value OR dipar.Kr2_ON.value) THEN 
	tau := 10.0;  ELSE tau := 100.0; 
END_IF;

IF NOT dipar.Kr5_off.value THEN p_in := 0.0;
ELSIF dipar.Kr6_ON.value AND am.Kr6.isOFF THEN p_in := Pg_in;
ELSIF dipar.Kr4_ON.value OR dipar.Kr1_ON.value THEN p_in := Pg_in;
END_IF;

IF tau < 100.0 THEN 
	aipar.Pg_inN.sim_value := aipar.Pg_inN.sim_value + (p_in - aipar.Pg_inN.value) / (tau);
	aipar.Pg_outN.sim_value := aipar.Pg_inN.sim_value + acpar.Nst.value * kx;
END_IF; 

dipar.Pg_outKR1.sim_value := aipar.Pg_inN.value > 2.6;

//dipar.SK_OF.sim_value	:= am.SK.isOFF;
//dipar.SK_ON.sim_value	:= am.SK.isON;

//Т газа
aipar.Tg_inN.sim_value := aipar.Tg_inN.sim_value + (aipar.Ta_inK.value + aipar.Pg_inN.value * 4.2 - aipar.Tg_inN.sim_value)/(tau_det);
aipar.Tg_outN.sim_value := aipar.Tg_outN.sim_value + (aipar.Ta_inK.value + aipar.Pg_outN.value * 4.2 - aipar.Tg_outN.sim_value)/(tau_det);

IF aipar.Pg_inN.value < 0 THEN aipar.Pg_inN.sim_value := 0; END_IF;
IF aipar.Pg_outN.value < 0 THEN aipar.Pg_outN.sim_value := 0; END_IF;

                  
END_FUNCTION

FUNCTION ALG_BN_link : BOOL

                    
subsystem.BN(
	sys_type := 1,
	work := acpar.Nst.value > 20.0, 
	stop := acpar.Nst.value <= 20.0);
	
ALG_BN_base();
                  
END_FUNCTION

///
/// Назначение: 		Формирование выходных сигналов для сторожевого таймера
/// Автор: 			
/// Версия: 			00.00.01
FUNCTION ALG_PLC : BOOL
VAR
	cycle : REAL := GVL_LIB.cycle_time_fast;
END_VAR

                    
//Формирование меандра для реле БЭО
plc.BEO(tau := T#200MS, T := T#400MS, cycle := cycle);
dopar.BEO_w1.value := dopar.BEO_w2.value := plc.BEO.out;
                  
END_FUNCTION

///
/// Назначение: 		Вызов подрежимов
/// Автор: 			
/// Версия: 			00.00.01
FUNCTION ALG_SMD_link : BOOL

                    
//Функция обработки режимов и подрежимов с шагами
smd_update(cycle := cycle_time_base);
                  
END_FUNCTION

///
/// Назначение: 		Формирование выходных сигналов, не входящих ни в одну группу
/// Автор: 			
/// Версия: 			00.00.01
FUNCTION ALG_AM : BOOL

                    
dopar.Sound_ON.value := HP.cmd_sound_ON OR KPK.cmd_sound_ON OR APK.cmd_sound_ON;


                  
END_FUNCTION

FUNCTION ALG_D_AM_base : BOOL
VAR
	KPVOpen	: BOOL;
END_VAR

                    
//am.KPV1.on	:= ( AOss.cmd_KPV15_ON OR AObs.cmd_KPV15_ON OR am.KPV1.on ) AND NOT alg.V_000;
//am.KPV5.on	:= am.KPV1.on;

// Заглушка, т.к. КПВ1,5 управляются АУП-10
KPVOpen	:= ( acpar.NtkPrived.value > Ntk_KPVClose AND acpar.NtkPrived.value < Ntk_KPV15Open );
// КПВ 1
am.KPV1.on	:= KPVOpen;
// КПВ 2
am.KPV2.on	:= ( Start_D.cmd_KPV_On OR NOss.cmd_KPV234_ON OR NObs.cmd_KPV234_ON OR AOss.cmd_KPV234_ON OR AObs.cmd_KPV234_ON OR am.KPV2.on OR alg.V_000 ) AND NOT Start_D.cmd_KPV234_Off;
// КПВ 3
am.KPV3.on	:= am.KPV2.on;
// КПВ 4
am.KPV4.on	:= am.KPV2.on;
// КПВ 5
am.KPV5.on	:= KPVOpen;

// ВНА
am.VNA.on	:= Start_D.cmd_VNA_On OR NObs.cmd_VNA_On OR NOss.cmd_VNA_On OR AObs.cmd_VNA_On OR AOss.cmd_VNA_On;
// Обогрев ВНА
engine.VNAheat( par_value := aipar.Ta_inK.value, par_brk := aipar.Ta_inK.flt );
am.VNA_heat.on	:= ( engine.VNAheat.out OR dipar.Ace_alr.value ) AND NOT mde.Repair ;

// Агрегат зажигания
engine.AZ_off(IN := Start_D.cmd_AZ_ON);
am.AZ.on	:= engine.AZ_off.Q;
                  
END_FUNCTION

FUNCTION ALG_D_AM_fast : BOOL

                    // Стопорный клапан
//alg.SK_tr	:= (Start_D.cmd_SK_On OR alg.SK_tr) AND NOT (alg.AO OR alg.NO);
//am.SK.on	:= alg.SK_tr;

am.SK.on	:= (Start_D.cmd_SK_On OR am.SK.on) AND NOT (alg.AO OR NOss.cmd_SK_Off OR NObs.cmd_SK_Off);
                  
END_FUNCTION

{region INFO}
(*
 Назначение:   Используется для обработки аналоговых параметров, передаваемых с ВУ
 Автор:        /Разработчик/ 08.08.2025 8:32:24
 Конфигуратор: v00.01.00
 Проект:       KA107
*)
{endregion}
FUNCTION tunpar_update : BOOL
VAR_INPUT
END_VAR
VAR
END_VAR

                    tunpar.setNst(enable_direct_update := TRUE); //Задание Nst
tunpar.setNtk(enable_direct_update := TRUE); //Задание Ntk
tunpar.rateNstBtn(enable_direct_update := TRUE); //Шаг Nst для РЧВ
tunpar.rateNtkBtn(enable_direct_update := TRUE); //Шаг Ntk для РЧВ
tunpar.setTm(enable_direct_update := TRUE); //Задание температуры маслосистемы
tunpar.T1_avom(enable_direct_update := TRUE); //Т1 ПИД АВОМ
tunpar.T2_avom(enable_direct_update := TRUE); //Т2 ПИД АВОМ
tunpar.K_avom(enable_direct_update := TRUE); //К ПИД АВОМ
tunpar.DZ_avom(enable_direct_update := TRUE); //Зона нечувствительности ПИД АВОМ
tunpar.setTmMBDN(enable_direct_update := TRUE); //Температура в маслобаке смазки
tunpar.setTmMBN(enable_direct_update := TRUE); //Температура в маслобаке уплотнений
tunpar.countStart(enable_direct_update := TRUE); //Количество пусков
tunpar.countNO(enable_direct_update := TRUE); //Количество НО
tunpar.countAO(enable_direct_update := TRUE); //Количество АО
tunpar.generalOpTime(enable_direct_update := TRUE); //Наработка суммарная
tunpar.workOpTime(enable_direct_update := TRUE); //Наработка на режиме

                  
END_FUNCTION

FUNCTION tmr_update : BOOL

                    tmr.crsPmStarter_20();
//tmr.crsNIgnition_10();
//tmr.crsNBoost_10();
tmr.KPV15_nOpen();
tmr.KPV15_wOpen();
tmr.KPV234_wOpen();
tmr.PNU_S_Off();
tmr.PNU_S_pumpH();
                  
END_FUNCTION

{region INFO}
(*
 Назначение:   Ручной вызов обработчиков дискретных ИМов в fast цикле
 Автор:        /chekmarev/ 17.04.2025
 Проект:       KA107
*)
{endregion}
FUNCTION am_update_fast : BOOL

                    
//Стопорный клапан
//Тип: 1x2
am.SK(
	DU_prm := alg.V_000,
	onSigFlt := dipar.SK_ON.flt,
	onSig := dipar.SK_ON.value,
	onSig_sim_on := dipar.SK_ON.sim_on,
	onSig_sim_value := dipar.SK_ON.sim_value,
	offSigFlt	:= dipar.SK_off.flt,
	offSig		:= dipar.SK_off.value,
	offSig_sim_on:= dipar.SK_off.sim_on,
	offSig_sim_value := dipar.SK_off.sim_value,
	onFlt := dopar.SK_ON.flt);
dopar.SK_ON.value := am.SK.onOUT;
//--------------------------------------------------------------------------

//ДГ
//Тип: а
am.DG(
	PosSigFlt := aipar.DG_pos.flt,
	SetFlt := aopar.DG_set.flt,
	pos := aipar.DG_pos.value,
	pos_sim_on := aipar.DG_pos.sim_on,
	pos_sim_value := aipar.DG_pos.sim_value);
aopar.DG_set.value := am.DG.set_out;

 // Управление КПВ1, 5
dopar.KPV15_ON.value := ( am.KPV1.onOUT OR am.KPV5.onOut ) AND ( am.KPV1.DU AND am.KPV5.DU ) OR (( AOss.cmd_KPV15_ON OR AObs.cmd_KPV15_ON OR dopar.KPV15_ON.value ) AND NOT alg.V_000 );
// -----------------------------------
                  
END_FUNCTION

FUNCTION check_modes : BOOL

                    // Рп: Контроль ГР
PPU.Check_GR.value := (btn.GR.out OR NObs.finish OR HP.finish OR KPK.finish) OR PPU.Check_GR.value AND NOT (btn.HR.out OR btn.Repair.out OR btn.Start.out OR btn.Cancel.out OR alg.AO);

// Рп: Контроль ХР
PPU.Check_HR.value := (btn.HR.out OR btn.GR.out OR NObs.finish OR NOss.finish OR HP.finish OR KPK.finish) OR PPU.Check_HR.value AND NOT (btn.Repair.out OR btn.Start.out OR btn.Cancel.out OR alg.AO);

//Рп: Предпусковая готовность
check.btn := btn.HP.out OR btn.KPK.out OR btn.APK.out;
tch.PrepareStart.value := (check.btn OR tch.PrepareStart.value) AND NOT (btn.Start.out OR btn.Cancel.out OR mde.Repair);
   IF btn.HP.out THEN check.ready := ENUM_ReadyToStart.HP;
ELSIF btn.KPK.out THEN check.ready := ENUM_ReadyToStart.KPK;
ELSIF btn.APK.out THEN check.ready := ENUM_ReadyToStart.APK;
ELSIF NOT tch.PrepareStart.value THEN check.ready := ENUM_ReadyToStart.OFF;
END_IF;

//Рп: Сигналы готовности
tch.ReadyHP.value := ((check.ready = ENUM_ReadyToStart.HP AND tch.PrepareStart.value AND Check_SAU.finish) OR tch.ReadyHP.value) AND NOT (NOT (mde.GR OR mde.HR) OR btn.Cancel.out);
tch.ReadyKPK.value := ((check.ready = ENUM_ReadyToStart.KPK AND tch.PrepareStart.value AND Check_SAU.finish) OR tch.ReadyKPK.value) AND NOT (NOT (mde.GR OR mde.HR) OR btn.Cancel.out);
tch.ReadyAPK.value := ((check.ready = ENUM_ReadyToStart.APK AND tch.PrepareStart.value AND Check_SAU.finish) OR tch.ReadyAPK.value) AND NOT (NOT (mde.GR OR mde.HR) OR btn.Cancel.out);
check.ReadytoSF := tch.ReadyHP.value OR tch.ReadyKPK.value OR tch.ReadyAPK.value;


//Рп: Контроль САУ
//Проверка при подготовке к пуску или по кнопке при "Нет активных режимов" или каждые 12 часов, но не на пусковых режимах
check.tmr12H ( IN := NOT check.tmr12H.Q );
tch.Check_SAU.value := Check_SAU.drm.active;
check.tmrCancelPrm ( IN := Check_SAU.drm.active );
//Контроль виброаппаратуры двигателя (ИВ-Д-ПФ)
crs.Vs_D_Av.alg_check 	:= tch.Check_SAU.value;
crs.Vsst_HH.alg_check	:= tch.Check_SAU.value;
crs.Vstk_HH.alg_check	:= tch.Check_SAU.value;
crs.BZA_alr.alg_check	:= tch.Check_SAU.value;
dopar.Vibr_ctrl.value 	:= (Check_SAU.cmd_check_VibD OR dopar.Vibr_ctrl.value) AND NOT ( crs.Vs_D_Av.signalization AND crs.Vsst_HH.signalization AND crs.Vstk_HH.signalization OR btn.Cancel.out );
dopar.BZA_ctrl.value	:= (Check_SAU.cmd_check_BZA OR dopar.BZA_ctrl.value) AND NOT ( crs.BZA_alr.signalization OR btn.Cancel.out );
//tch.brk_vib_d.value := Check_SAU.cmd_check_VibD AND NOT (crs.VsPOD_OH.out AND crs.VsZOD_OH.out AND crs.VsD_Av.out);
//Разрешение старта
check.prm_start := (Check_SAU.finish AND check.ReadytoSF OR check.prm_start) AND NOT (btn.Start.out OR btn.Cancel.out OR mde.Repair);

//Имитация подрежима "Контроль САУ"
IF imitGPA.imit_on THEN check_imit(); END_IF;


                  
END_FUNCTION

FUNCTION check_imit : BOOL
VAR CONSTANT
	Ntk	: REAL := 8000;
END_VAR

                    check.tmrImit(IN := dopar.Vibr_ctrl.value OR dopar.BZA_ctrl.value);

dipar.Vs_D_Av.sim_value := check.tmrImit.Q;
dipar.BZA_alr.sim_value := check.tmrImit.Q;

aipar.Vstk.sim_value	:= TO_BYTE( check.tmrImit.Q ) * 92.0 + TO_REAL( SHR( PRG_base.result_time, 8) AND 2#00011111 ) * ( acpar.Ntk.value / Ntk );
aipar.Vsst.sim_value	:= aipar.Vstk.value;
                  
END_FUNCTION

FUNCTION_BLOCK TAcparHandler
VAR_INPUT
	/// в секундах 
	cycle: REAL;
END_VAR
VAR
	/// обработчики частот вращения 
	nTKfilter1: TMedianLagFilter;
	nTKfilter2: TMedianLagFilter;
	nSTfilter1: TMedianLagFilter;
	nSTfilter2: TMedianLagFilter;
	nTKcalc: TFreqRotorHandler;
	nSTcalc: TFreqRotorHandler;
END_VAR
VAR_TEMP
	// Среднее алгебраическое значение температуры
	TstAverage: REAL;
	// Количество исправных каналов
	TstCount: BYTE;	
END_VAR

                    (* фильтрация оборотов *)
(* нулевая постоянная времени фильтра тут корректна, при этом остается только медианный фильтр (чтобы убрать одиночные выбросы). 
При надобности можно увеличить tau, если нужен фильтр высокочастотной помехи (не отдельные "шилья", а "борода" на сигнале) *)
nTKfilter1( inVal:= aipar.Ntk_1.value, inBrk:= aipar.Ntk_1.flt, tau:= 0.3, cycle:= cycle ); 
nTKfilter2( inVal:= aipar.Ntk_2.value, inBrk:= aipar.Ntk_2.flt, tau:= 0.3, cycle:= cycle ); 
nSTfilter1( inVal:= aipar.Nst_1.value, inBrk:= aipar.Nst_1.flt, tau:= 0.3, cycle:= cycle ); 
nSTfilter2( inVal:= aipar.Nst_2.value, inBrk:= aipar.Nst_2.flt, tau:= 0.3, cycle:= cycle ); 

(* обработка двойных датчиков оборотов *)
nTKcalc.ch[1] 	:= nTKfilter1.outVal;
nTKcalc.ch[2]	:= nTKfilter2.outVal;
nTKcalc( disbal_Ch := 100.0, maxVal := aipar.Ntk_1.cfg.hilim, minVal := 100.0, ucvV := 500, flt_prm := acpar.Ntk.value > 500.0, deblock := btn.Unlock.out, out := acpar.Ntk );

nSTcalc.ch[1] 	:= nSTfilter1.outVal;
nSTcalc.ch[2]	:= nSTfilter2.outVal;
nSTcalc( disbal_Ch := 100.0, maxVal := aipar.Nst_1.cfg.hilim, minVal := 100.0, ucvV := 500, flt_prm := acpar.Nst.value > 500.0, deblock := btn.Unlock.out, out := acpar.Nst );

// обработка кольца термопар
{warning ' Убедиться, что в настройках модулей UCP1_A1_AI6 и UCP1_A1_AI7 выставлены диапазоны на каналах термопар (-50...+800) '}
// flt от модуля - обрыв или выход за пределы диапазона температур (-50...+800)
//TstCount := 0;
IF ( NOT aipar.Tg_inST_1.flt ) THEN
	TstAverage 	:= aipar.Tg_inST_1.value;
	TstCount 	:= 1;
END_IF
IF ( NOT aipar.Tg_inST_2.flt ) THEN
	TstAverage 	:= TstAverage + aipar.Tg_inST_2.value;
	TstCount	:= TstCount + 1;
END_IF
IF ( NOT aipar.Tg_inST_3.flt ) THEN
	TstAverage 	:= TstAverage + aipar.Tg_inST_3.value;
	TstCount	:= TstCount + 1;
END_IF
IF ( NOT aipar.Tg_inST_4.flt ) THEN
	TstAverage 	:= TstAverage + aipar.Tg_inST_4.value;
	TstCount	:= TstCount + 1;
END_IF
IF ( NOT aipar.Tg_inST_5.flt ) THEN
	TstAverage 	:= TstAverage + aipar.Tg_inST_5.value;
	TstCount	:= TstCount + 1;
END_IF
IF ( NOT aipar.Tg_inST_6.flt ) THEN
	TstAverage 	:= TstAverage + aipar.Tg_inST_6.value;
	TstCount	:= TstCount + 1;
END_IF

acpar.Tg_inST.flt 	:= TstCount = 0;
alg.TstInWork		:= TstCount;

IF TstCount > 0 THEN
	acpar.Tg_inST.in_value	:= TstAverage / TstCount;	
END_IF

(* все полученные данные выкладываются на входы acpar, acpar обновляются в своей автоматически сформированной функции *)
//acpar.Ntk.in_value := nVDcalc.value; acpar.Ntk.flt := nVDcalc.disbalanse;
//acpar.Nst.in_value := nSTcalc.value; acpar.Nst.flt := nSTcalc.disbalanse;
IF NOT aipar.Ta_inK.flt THEN acpar.NtkPrived.in_value := acpar.Ntk.value * SQRT( 288.15 / ( aipar.Ta_inK.value + 273.15 ) );
ELSE acpar.NtkPrived.in_value := acpar.Ntk.value;
END_IF;
acpar.Qtg_m3.in_value := FuelReg.fReg.fuel; 
                  
END_FUNCTION_BLOCK

FUNCTION_BLOCK TMedianLagFilter
VAR_INPUT
	inVal: REAL;
	inBrk: BOOL;
	tau: REAL;
	cycle: REAL;
END_VAR
VAR_OUTPUT
	outVal: REAL := 0;
END_VAR
VAR
	inArr: ARRAY[0..2] OF REAL;
	idx: INT := 0;
	cnt: INT;
	minVal: REAL := 1000000;
	maxVal: REAL := -1000000;
	sum: REAL;
END_VAR

                    IF inBrk THEN
	outVal := 0.0;
ELSE
  // заполнить входной массив, работает как кольцевой буфер
  inArr[ idx ] := inVal;
  idx := idx + 1;
  IF idx > 2 THEN idx := 0; END_IF;
  // сразу найти сумму - закладка под бОльщую размерность массива
  sum := 0.0;
  minVal := 1000000.0;
  maxVal := -1000000.0;
  FOR cnt := 0 TO 2 DO
	sum := sum + inArr[cnt];
    IF inArr[cnt] > maxVal THEN maxVal := inArr[cnt]; END_IF;  
    IF inArr[cnt] < minVal THEN minVal := inArr[cnt]; END_IF;  
  END_FOR
  // отбраковать минимум, максимум
  sum := sum - maxVal - minVal;
  // инерционное звено
  IF tau > cycle THEN
    outVal := outVal + ( cycle / tau ) * ( sum - outVal );	
  ELSE
	outVal := sum;   
  END_IF; 	
END_IF

                  
END_FUNCTION_BLOCK

FUNCTION FR_link : BOOL

                    // заполнение входных полей типа 
FuelReg.fReg.Nvd.value := acpar.Ntk.value; 
FuelReg.fReg.Nst.value:= acpar.Nst.value; 
FuelReg.fReg.Tg_outST.value:= acpar.Tg_inST.value; 
FuelReg.fReg.Pa_K.value:= aipar.Pa_out14.value; 
FuelReg.fReg.Ta_inD.value:= aipar.Ta_inK.value; 
FuelReg.fReg.Ttg_inValve.value := aipar.Ttg.value;
FuelReg.fReg.Ptg_inValve.value := aipar.Ptg_inTRK.value;
FuelReg.fReg.Nvd.flt := acpar.Ntk.flt; 
FuelReg.fReg.Nst.flt:= acpar.Nst.flt; 
FuelReg.fReg.Tg_outST.flt:= acpar.Tg_inST.flt; 
FuelReg.fReg.Pa_K.flt:= aipar.Pa_out14.flt; 
FuelReg.fReg.Ta_inD.flt:= aipar.Ta_inK.flt; 
FuelReg.fReg.Ttg_inValve.flt := aipar.Ttg.flt;
FuelReg.fReg.Ptg_inValve.flt := aipar.Ptg_inTRK.flt;

// обновление настроек
FuelRegTuns_update();

FuelReg.fReg(
	calcStep:= cycle_time_fast, 
    setValNvdExt:= tunpar.setNtk,  
	setValNstExt:= tunpar.setNst, 
	//startCom:= , // пишется в последовательностях
	checkCom := crs.Fire_flt.check,
    normalStopCom:= alg.normalStopCom, 
	emergStopCom:= alg.emergStopCom, 
	regNstOn:= bn.stabSTbtn, 
	fuel=>acpar.Qtg_m3.in_value, 
	setValve=>am.DG.set, 
	//start=> , // читается в последовательностях
	//heating=> , 
	//started=> , 
	//cooling=> , 
	//stoped=> , 
	//heatCountdown=> , 
	//coolCountdown=> , 
	//isFire=> 
     );
	 
FuelReg.fReg.update();	 


                  
END_FUNCTION

///
/// Назначение: 		Программный имитатор
/// Автор: 			
/// Версия: 			00.00.01
FUNCTION imit : BOOL
VAR CONSTANT
	tm: REAL := 15;
END_VAR

                    
//Инициализация
IF imitGPA.init (* OR testing.init *)THEN
	
	aipar.Tm_inD.sim_value	:= tm;
	aipar.Tm_MB.sim_value	:= tm;
	aipar.Tm_MBU.sim_value	:= tm;
	aipar.Tm_outAU.sim_value:= tm;
	aipar.Tm_outD.sim_value	:= tm;
	aipar.Tm_outAVOM.sim_value:= tm;
	
	aipar.Ta_inK.sim_value	:= tm;
	aipar.Tg_inST_1.sim_value := tm;
	aipar.Tg_inST_2.sim_value := tm + 2.3;
	aipar.Tg_inST_3.sim_value := tm - 1.2;
	aipar.Tg_inST_4.sim_value := tm;
	
	dipar.BZA_ready_1.sim_value		:= TRUE;
	dipar.Fuse_AO_UCP1.sim_value 	:= TRUE;
	dipar.Fuse_DO_UCP1.sim_value 	:= TRUE;
	dipar.Fuse_Air_UCP1.sim_value	:= TRUE;
	dipar.Fuse_DO_UE1.sim_value		:= TRUE;
	dipar.U_main.sim_value			:= TRUE;
	dipar.U_res.sim_value			:= TRUE;
	dipar.AG1.sim_value				:= TRUE;
	dipar.AG2.sim_value				:= TRUE;
	dipar.AG3.sim_value				:= TRUE;
	dipar.AG4.sim_value				:= TRUE;
	dipar.AG10.sim_value			:= TRUE;
	dipar.AG15.sim_value			:= TRUE;
	dipar.AG16.sim_value			:= TRUE;
	dipar.AG5.sim_value				:= TRUE;
	dipar.AG6.sim_value				:= TRUE;
	dipar.AG8.sim_value				:= TRUE;
	dipar.AG9.sim_value				:= TRUE;
	dipar.AG17.sim_value			:= TRUE;
	dipar.AG18.sim_value			:= TRUE;
	dipar.U_PRU.sim_value			:= TRUE;
	dipar.Utrk_main.sim_value		:= TRUE;
	dipar.U_AI.sim_value			:= TRUE;
	dipar.U_DI.sim_value			:= TRUE;
	dipar.U_BIZ.sim_value			:= TRUE;
	dipar.U_AM.sim_value			:= TRUE;
	dipar.Uvs_24.sim_value			:= TRUE;
	dipar.Uother_24.sim_value		:= TRUE;
	dipar.U_AM2.sim_value			:= TRUE;
	dipar.Utrk_res.sim_value		:= TRUE;
	dipar.Ubeo_main.sim_value		:= TRUE;
	dipar.Ubeo_res.sim_value		:= TRUE;
	dipar.AG11.sim_value			:= TRUE;
	dipar.AG12.sim_value			:= TRUE;
	dipar.U_KEAO.sim_value			:= TRUE;
	dipar.U_BEO.sim_value			:= TRUE;
	dipar.U_BZA.sim_value			:= TRUE;
	dipar.TRKready.sim_value		:= TRUE;
	
	dipar.EV1.sim_value				:= FALSE;
	dipar.EV2.sim_value				:= FALSE;
	dipar.EV3.sim_value				:= FALSE;
	dipar.EV4.sim_value				:= FALSE;
	dipar.Err_AUO1.sim_value		:= FALSE;
	
	dipar.Lm_MB_Pn.sim_value		:= FALSE;

	dipar.Lm_MBU_Pn.sim_value		:= FALSE;
	dipar.AO_PRU_2.sim_value		:= FALSE;
	dipar.Ace_alr.sim_value			:= FALSE;
	
	//Краны в положение останова
	am.Kr1.off 	:= TRUE;
	am.Kr2.off 	:= TRUE;
	am.Kr4.off 	:= TRUE;
	am.Kr5.on 	:= TRUE;	
	am.Kr6.off 	:= TRUE;
	am.Kr9.on 	:= TRUE;
	am.Kr10.on 	:= TRUE;
	am.Kr11.off := TRUE;
	am.Kr12.off := TRUE;
	am.KR13.off := TRUE;
	am.Kr15.off := TRUE;

	btn.Unlock.cmd := TRUE;
	imitGPA.init := FALSE;
END_IF;

IF imitGPA.imit_on THEN
	fun_ACS();
END_IF

//Включение имитации
imitGPA.imit_on := btn.imit_ON.out OR GVL_LIB.isTrainer OR imitGPA.imit_on AND NOT (btn.imit_OF.out);
gvl_lib.sim_on_all := imitGPA.imit_on;

//Переиницализация параметров начальными значениями при входе в имитацию
imitGPA.imit_start(CLK := imitGPA.imit_on);
imitGPA.init := imitGPA.imit_start.Q;
                  
END_FUNCTION

FUNCTION_BLOCK TImitEngineTuns
VAR_INPUT
	/// таблица открытия 
	openToGt: TLinear;
	GtToNvd: TLinear;
	GtToTst: TLinear;
	NvdToTauNvd: TLinear;
	NvdToTauTst: TLinear;
	NvdToTauPk: TLinear;
	NstToTauNst: TLinear;
	NvdToTst: TLinear;
	NvdToPk: TLinear;
	NvdToNst: TLinear;
	DUSdz: REAL;
	DUSrate: REAL;
	NvdStart: REAL;
END_VAR

                    
                  
END_FUNCTION_BLOCK

///2023-05-20
FUNCTION_BLOCK TEngineModel
VAR_INPUT
	/// температура атмосферного воздуха, ∞C
	Tatm: REAL;
	/// задание на ДГ, %
	setDG1: REAL;
	/// задание на ДГ, %
	setDG2: REAL;
	/// задание на ВНА, ∞
	setVNA: REAL;
	/// задание на  КПВ, ∞
	setKPV: REAL;
	/// призак работы стартера
	starter: BOOL;
	/// длЯ электростартера - работа на первой скорости
	starterSpeed1: BOOL;
	/// служебные сигналы, задающие конфигурацию ГТУ: наличие роторов среднего
	SDpresent: BOOL;
	/// и низкого давлениЯ газогенератора,
	NDpresent: BOOL;
	/// необходимость моделированиЯ давлениЯ за компрессором,
	PkPresent: BOOL;
	/// наличие дополнительного дозатора топлива,
	DUSaddPresent: BOOL;
	/// электростартер (по умолчанию - турбостартер)
	elStart: BOOL;
	cycle: REAL := cycle_time_fast;
	/// шаг интегрированиЯ в секундах 
	step: REAL;
	tuns: POINTER TO TImitEngineTuns;
END_VAR
VAR_OUTPUT
	/// расход топлива (кг/ч)
	Gfuel: REAL;
	/// положение ƒ√1, %
	posDG1: REAL;
	/// положение ƒ√1, %
	posDG2: REAL;
	/// положение ¬Ќј, ∞
	posVNA: REAL;
	/// положение  ѕ¬, ∞
	posKPV: REAL;
	/// частота вращения  Ќƒ, об/мин
	Nnd: REAL;
	/// среднего давлениЯ
	Nsd: REAL;
	/// частота вращения  ¬ƒ, об/мин
	Nvd: REAL;
	/// частота вращения —“, об/мин
	Nst: REAL;
	/// температура за “Ќƒ, ∞C
	Tt: REAL;
	/// температура за —“, ∞C
	Tst: REAL;
	/// давление за компрессором, ћѕа
	Pk: REAL;
	/// мощность двигателЯ в кВт
	power: REAL;
END_VAR
VAR
	/// зона нечувствительности привода ДУС (в %)
	DUS_DZ: REAL;
	/// скорость перемещениЯ привода ДУС (в %/с)
	DUS_RATE: REAL;
	NvdStart: REAL;
	/// расход топлива приведенный (кг/ч)
	Gt0: REAL;
	/// приведеннаЯ частота вращениЯ ротора ВД
	nvd0: REAL;
	/// частота вращениЯ ротора ВД, развиваемаЯ при раскрутке стартером
	NvdSetStarter: REAL;
	/// установившеесЯ значение частоты вращениЯ ротора ВД  
	nVDset: REAL;
	/// установившеесЯ значение температуры продуктов сгораниЯ перед СТ
	tSTset: REAL;
	tSTtoTT: REAL;
	/// количество шагов интегрированиЯ
	stepQuantity: DINT;
	/// счетчик шагов интегрированиЯ
	integCount: DINT;
	init: BOOL := FALSE;
	/// температура за ГГ на установившемся режиме
	Tt0: REAL;
END_VAR

                    IF NOT init THEN // инициализациЯ - производитсЯ считывание настроек, модель устанавливаетсЯ в нулевое начальное состоЯние
    DUS_DZ        := tuns^.DUSdz;
    DUS_RATE      := tuns^.DUSrate; 
    NvdStart := tuns^.NvdStart;
	tSTtoTT := 1.35; 
    Gt0  := 0.0;
    nvd0 := 0.1;
    NvdSetStarter := tuns^.NvdStart;
    nVDset := 0.1;
    tSTset := 0.0;
    posDG1 := 0.0;
    posDG2 := 0.0;
    nsd := 0.0;
    nnd := 0.0;
    nst := 0.0;
    init:= true;
    stepQuantity := REAL_TO_DINT(cycle/step + 0.5);
  ELSE // основнаЯ работа
    FOR integCount := 1 TO stepQuantity DO 
      // моделирование привода ДУСа (основного и дополнительного)
      // дозаторы топлива имеют шаговый электропривод с высоким быстродействием.
      IF nvd0 < 0.1 THEN nvd0 := 0.1; END_IF;
// Упрощаем имитацию ДУСа
//      DUSmdl(set := setDUSmain, dz := 0.25, cycle := step); 
      //YDUSmain := DUSmdl.out;
//      YDUSmain := setDUSmain;
      IF ABS( setDG1 - posDG1 ) > DUS_DZ THEN
        posDG1 := posDG1 + (step/( 0.3 * 100.0 / tuns^.DUSrate ) ) * (setDG1 - posDG1);		  
      END_IF;   
(* 
      IF setDG1 - posDG1 > DUS_DZ THEN
        posDG1 := posDG1 + step*DUS_RATE;
        IF posDG1 > setDG1 THEN posDG1 := setDG1; END_IF;
      ELSIF setDG1 - posDG1 < -DUS_DZ THEN
        posDG1 := posDG1 -step*DUS_RATE;
        IF posDG1 < setDG1 THEN posDG1 := setDG1; END_IF;
      END_IF;
      // длЯ двухзонных камер сгораниЯ: многозонность горениЯ не учитываетсЯ, а просто учитываетсЯ суммарный расход 
      //топлива через два дозатора
      IF DUSaddPresent THEN
        IF setDG2 - posDG2 > DUS_DZ THEN
          posDG2 := posDG2 + step*DUS_RATE;
          IF posDG2 > setDG2 THEN posDG2 := setDG2; END_IF;
        ELSIF setDG2 - posDG2 < -DUS_DZ THEN
          posDG2 := posDG2 -step*DUS_RATE;
          IF posDG2 < setDG2 THEN posDG2 := setDG2; END_IF;
        END_IF;
      END_IF;
      *)
	  tuns^.openToGt( arg := posDG1 + posDG2 );
      Gt0 := (tuns^.openToGt.out) * TO_INT(NOT dipar.SK_off.value);
      
      tuns^.GtToNvd(arg := Gt0 );
      tuns^.NvdToTauNvd(arg := Nvd);

      IF Gt0 < 0.0 THEN Gt0 := 0.0; END_IF;
  //    IF DUSaddPresent THEN Gt0 := Gt0 + tunings(tunName := tunConst.YDUSaddToGt, arg := YDUSadd); END_IF;
      // расход топлива
      // момент стартера
      IF starter THEN
        IF elStart THEN
          IF starterSpeed1 THEN NvdSetStarter := NvdStart/ 2.0;
          ELSE NvdSetStarter := NvdStart; END_IF;              
          // добавлено моделирование различной мощности электростартера на первой и второй скорости 
          IF NvdSetStarter > tuns^.GtToNvd.out THEN 
            nVDset := NvdSetStarter;
          ELSE nVDset := tuns^.GtToNvd.out;
          END_IF;       
        ELSE    
          nVDset := NvdStart + tuns^.GtToNvd.out;
        END_IF;  
      ELSE    
        nVDset := tuns^.GtToNvd.out;    
      END_IF;  
      // электростартер имеет почти постоЯнные обороты, поэтому обгоннаЯ муфта его
      // отключает. Турбостартер передает момент на вал всегда, когда включен
      // зубчатой муфтой и к нему подведен пусковой газ
      nvd0 := nvd0 + (step/(tuns^.NvdToTauNvd.out+0.001)) * (nVDset - nvd0);
      // частота вращениЯ ротора высокого давлениЯ (приведеннаЯ)
	  
      tuns^.GtToTst(arg := Gfuel);
      tuns^.NvdToTst(arg := Nvd);
      tuns^.NvdToTauTst(arg := Nvd);
	  
      tSTset := Tatm + tuns^.GtToTst.out - tuns^.NvdToTst.out;
	  IF tSTset < 0.0 THEN tSTset := 0.0; END_IF;
      Tst := Tst + (step/tuns^.NvdToTauTst.out) * (tSTset - Tst);
      // температура продуктов сгораниЯ вычислЯетсЯ в зависимости от частоты вращениЯ (-) и расхода топлива (+), учитываетсЯ
 
      Tt0 := tuns^.GtToTst.out - tuns^.NvdToTst.out;
      Tt  := Tt + (Tt0 - Tt) / tuns^.NvdToTauTst.out * cycle;

     // динамика
      nvd := nvd0 * SQRT((273.15 + Tatm)/288.15);
   (*   IF NDpresent THEN
        IF SDpresent THEN
          nsd := nsd + (step/(tunings(tunName := tunConst.nsdToTauSD, arg := nsd)+0.001))*
            (tunings(tunName := tunConst.nvdToNsd, arg := nvd) - nsd);
          nnd := nnd + (step/(tunings(tunName := tunConst.nndToTauND, arg := nnd)+0.001))*
            (tunings(tunName := tunConst.nsdToNnd, arg := nsd) - nsd);
        ELSE
          nsd := 0.0;
          nnd := nnd + (step/(tunings(tunName := tunConst.nsdToTauSD, arg := nnd)+0.001))*
            (tunings(tunName := tunConst.nvdToNsd, arg := nvd) - nnd); 
        END_IF;  
      END_IF;  
      // такаЯ хитраЯ логика свЯзана с терминологией: на двухвальных газогенераторах есть роторы ВД и НД, а на трехвальных - 
      // ВД, СД и НД. Поэтому, при наличии только флага НД игнорируетсЯ СД, а НД вычислЯетсЯ как СД.
	  *)	  	  
      IF PkPresent THEN
		tuns^.NvdToPk(arg := Nvd);
        tuns^.NvdToTauPk(arg := Nvd);
        Pk := Pk + (step/(tuns^.NvdToTauPk.out + 0.001)) * (tuns^.NvdToPk.out - Pk);
      END_IF;        
	  
	  
      (* пока не нужно, пригодится для генератора  
      power := tunings(tunName := tunConst.nvdToPower, arg := nvd0);
	  *)
      Gfuel := Gt0;
      // А здесь скорость СТ подсчитаем по упрощённой модели
 	  tuns^.NvdToNst(arg := Nvd);
      tuns^.NstToTauNst(arg := Nst);
      nst := nst + (step/(tuns^.NstToTauNst.out+0.001))*
                         (tuns^.NvdToNst.out - nst);
    END_FOR;
  END_IF; 	
	
	
                  
END_FUNCTION_BLOCK

FUNCTION_BLOCK TEdgeDetect
VAR_INPUT
	/// Вход импульсов
	in: BOOL;
END_VAR
VAR
	/// Передний край
	fe: BOOL;
	/// Задний край	
	re: BOOL;
	/// Предыдущее состояние входа
	oldin: BOOL;
	/// Промежуточное значение
	z: BOOL;
	/// Триггер переднего фронта 
	tf: BOOL;
	/// Триггер заднего фронта
	tr: BOOL;
END_VAR

                    z	:= in XOR oldIn;
fe	:= z AND in;
re	:= z AND oldin;
oldin := in;

tf	:= fe OR tf;	// tf и tr сбрасываем в акцессоре
tr	:= re OR tr;
                  

/// Выделение переднего фронта
PROPERTY Qf : BOOL
GET
                            Qf	:= tf;
tf	:= false;
                          
END_GET
SET
PRIVATE
                            
                          
END_SET
END_PROPERTY

/// Выделение заднего фронта
PROPERTY Qr : BOOL
GET
                            Qr	:= tr;
tr	:= false;
                          
END_GET
SET
PRIVATE
                            
                          
END_SET
END_PROPERTY
END_FUNCTION_BLOCK

FUNCTION ALG_BN_base : BOOL

                    // РЧВ
IF btn.turnDN.Qf THEN
	tunpar.setNst.set_value := tunpar.setNst.value - tunpar.rateNstBtn.value * TO_BYTE ( bn.stabSTbtn );
	tunpar.setNtk.set_value := tunpar.setNtk.value - tunpar.rateNtkBtn.value * TO_BYTE ( NOT bn.stabSTbtn );	
END_IF

IF btn.turnUP.Qf THEN
	tunpar.setNst.set_value := tunpar.setNst.value + tunpar.rateNstBtn.value * TO_BYTE ( bn.stabSTbtn );
	tunpar.setNtk.set_value := tunpar.setNtk.value + tunpar.rateNtkBtn.value * TO_BYTE ( NOT bn.stabSTbtn );
END_IF

IF NOT bn.stabSTbtn OR NOT tch.GTDwork.value THEN
	tunpar.setNst.value := acpar.Nst.value;
END_IF

IF bn.stabSTbtn OR NOT tch.GTDwork.value THEN
	tunpar.setNtk.value := acpar.Ntk.value;
END_IF

// Вытяжной вентилятор контейнера
am.VVN.on := dipar.Zagaz_OD_Pv.value;
bn.VVN_OFF( IN := NOT dipar.Zagaz_OD_Pv.value );
am.VVN.off:= bn.VVN_OFF.Q;
                  
END_FUNCTION

/// Маслоохладитель с дискретным включением вентиляторов
/// Вентиляторы включаются по наименьшей наработке
/// Выключаются - по наибольшей
/// Chekmarev
FUNCTION_BLOCK TAVOM
VAR_INPUT
	// разрешение работы АВОМ
	enable	: BOOL;
END_VAR
VAR_IN_OUT
	// Уставка температуры в маслосистеме
	Tm_SET	: Ttunpar;
	// Уставка Т1 для ПИД
	T1		: Ttunpar;
	// Уставка Т2 для ПИД
	T2		: Ttunpar;
	// Уставка K для ПИД
	K		: Ttunpar;
	// Уставка DZ для ПИД
	DZ		: Ttunpar;
	// Первый вентилятор маслоохладителя
	Vn1_AVOM: TAM_2x1;
	// Второй вентилятор маслоохладителя
	Vn2_AVOM: TAM_2x1;
	// Третий вентилятор маслоохладителя
	Vn3_AVOM: TAM_2x1;
	// Четвёртый вентилятор маслоохладителя
	Vn4_AVOM: TAM_2x1;	
END_VAR
VAR
	/// массив указателей на вентиляторы
	Vn_s: ARRAY[1..4] OF POINTER TO TAM_1x1;
	/// таймер отсчёта периода импульса
	tmrT: TON;
	/// Значение таймера на предыдущем цикле
	tmrT_Qold: BOOL;
	/// регулятор температуры масла
	TmReg: TPID;
	///	TmImp		: TP;		// инкремент / декремент счётчика
	///	target		: REAL;	
	_dz: REAL := 10;
	/// Флаг-указание на включение вентилятора из очереди
	_On: BOOL;
	/// Флаг-указание на отключение вентилятора из очереди
	_Off: BOOL;
END_VAR

                    
Vn_s[1]	:= ADR ( Vn1_AVOM );
Vn_s[2]	:= ADR ( Vn2_AVOM );
Vn_s[3]	:= ADR ( Vn3_AVOM );
Vn_s[4]	:= ADR ( Vn4_AVOM );
                  

METHOD PRIVATE PIDreg : BOOL
VAR_INPUT
	/// регулируемая температура
	temperature	: REAL;
END_VAR
VAR
	/// Ошибка регулирования	
	dTm: REAL;
END_VAR
                          // Регулирование с нуля
IF enable THEN
	TmReg.set_tun := FALSE;
	ELSE
		TmReg.set_tun	:= TRUE;
		TmReg.integ_tun	:= 0;
		TmReg.out_tun	:= 0;
END_IF

dTm := temperature - Tm_SET.value;

TmReg.setPID(_K := K.value, _T1 := T1.value, _T2 := T2.value, _DZ := DZ.value);
TmReg.singlePID(	err 	:= dTm,
					hiLimit	:= 100,
					loLimit	:= -100,
					hiRate	:= 10,
					loRate	:= 10,
					cycle	:= cycle_time_base,
					setDU	:= 0,
					DU		:= FALSE);
					
//target := TmReg.out;
                        
END_METHOD

/// Вентиляторы маслоохладителя
METHOD PRIVATE VnCntrl : BOOL
VAR
	index	: BYTE;
	min_	: BYTE := 1;
	max_	: BYTE := 1;
	on_1	: BOOL := TRUE;
	off_1	: BOOL := TRUE;
END_VAR
                          FOR index := 1 TO 4 DO
	Vn_s[index]^.on 	:= Vn_s[index]^.notOn AND Vn_s[index]^.flt;
	Vn_s[index]^.off 	:= FALSE;
END_FOR

IF On THEN
	FOR index := 1 TO 4 DO
	IF Vn_s[index]^.DU OR Vn_s[index]^.on THEN CONTINUE; END_IF
	IF Vn_s[index]^.isOFF THEN
		IF on_1 THEN
			min_ := index;
			on_1 := FALSE;
		END_IF
		IF Vn_s[index]^.OperationTime <= Vn_s[min_]^.OperationTime THEN
			min_ := index;
		END_IF
	END_IF
	END_FOR
	
	Vn_s[min_]^.off:= FALSE;
	Vn_s[min_]^.on := NOT Vn_s[min_]^.isON;
END_IF

IF Off THEN
	FOR index := 1 TO 4 DO
	IF Vn_s[index]^.DU OR Vn_s[index]^.off THEN CONTINUE; END_IF
	IF Vn_s[index]^.setOn THEN
		IF off_1 THEN
			max_ := index;
			off_1 := FALSE;
		END_IF
		IF ( Vn_s[index]^.OperationTime >= Vn_s[max_]^.OperationTime ) THEN
			max_ := index;
		END_IF
	END_IF
	END_FOR
	
	Vn_s[max_]^.on	:= FALSE;
	Vn_s[max_]^.off := Vn_s[max_]^.setOn; //NOT Vn_s[max_]^.isOFF OR Vn_s[max_]^.notOn;
END_IF
                        
END_METHOD

/// Chekmarev
METHOD update : BOOL
VAR_INPUT
	// регулируемая температура
	temperature	: REAL;
END_VAR
VAR
	// период следования импульсов
	T: TIME := TIME#1m0s0ms;
END_VAR
                          
PIDreg(temperature := temperature);

// Шаг импульса зависит от величины коррекции ошибки ПИД регулятором
// ( реализация ЧИМ )
T := TO_TIME (( 110 - ABS ( TmReg.out )) * 1000 );

tmrT ( in := NOT tmrT.Q, PT := T );

// Выделяем передний фронт импульса выхода таймера
IF (( tmrT.Q XOR tmrT_Qold ) AND tmrT.Q ) THEN
	IF ( 0 < tmreg.out - _DZ ) THEN
		_On 	:= TRUE;	// снимается в акцессоре
		_Off	:= FALSE;	// снимем на всякий случай
	END_IF
	
	IF ( 0 >= tmreg.out + _DZ ) THEN
		_On		:= FALSE;	// снимем на всякий случай
		_Off	:= TRUE;	// снимается в акцессоре
	END_IF
END_IF

tmrT_Qold := tmrT.Q;

IF NOT enable THEN
	_On	:= FALSE;
	_Off:= TRUE;
END_IF

VnCntrl();
                        
END_METHOD

/// Необходимо включить очередной вентилятор
PROPERTY On : BOOL
GET
PRIVATE
                            On		:= _On;
_On 	:= FALSE;
                          
END_GET
SET
PRIVATE
                            
                          
END_SET
END_PROPERTY

/// Необходимо выключить очередной вентилятор
PROPERTY Off : BOOL
GET
PRIVATE
                            Off		:= _Off;
_Off 	:= FALSE;
                          
END_GET
SET
PRIVATE
                            
                          
END_SET
END_PROPERTY
END_FUNCTION_BLOCK

PROGRAM PRG_PRU_Base
VAR_INPUT
	
	General: ARRAY[0..1] OF WORD := [4, 0];	/// номер агрегата [0] и режимх[1] 
	Holdings: ARRAY[0..16] OF REAL;
	Coils: ARRAY[0..13] OF BYTE;
	StatusReal: WORD;
END_VAR
VAR	
	Count: BYTE;	/// счётчик ошибок связи с ПРУ
	LinkPSU: BOOL;
	LinkPSUold: BOOL;
END_VAR

                    // Контроль связи с ПСУ
LinkPSU	:= Coils[13].1 XOR Coils[13].0;
IF LinkPSU THEN
	Count := Count + 1;
	ELSE
	Count := 0;
	PRU.Link := TRUE;
	LinkPSUold		:= NOT LinkPSUold;
END_IF

IF Count > 254 THEN 
	PRU.Link 	:= FALSE; 
	Count 		:= 1;
//	LinkPSUold		:= NOT LinkPSUold;
END_IF;

Coils[13].0	:= LinkPSUold;

// Кнопки
btn.AOss.cmd_PRU	:= Coils[0].0;//btn_AOss_Кнопка "АОсс"
btn.AObs.cmd_PRU	:= Coils[0].1;//btn_AObs_Кнопка "АОбс"
btn.NOss.cmd_PRU	:= Coils[0].2;//btn_NOss_Кнопка "НОсс"
btn.NObs.cmd_PRU	:= Coils[0].3;//btn_NObs_Кнопка "НОбс"
btn.turnUP.cmd_PRU	:= Coils[0].4;//btn_turnUP_Кнопка "Увеличить обороты"
btn.turnDN.cmd_PRU	:= Coils[0].5;//btn_turnDN_Кнопка "Уменьшить обороты"

//Coils[0].6;//btn_regNvd_Кнопка "Регулирование оборотов ВД"
//Coils[0].7;//btn_regNst_Кнопка "Регулирование оборотов СТ"
//Coils[1].0				:= btn.AOss_PRU;//prm_AOss_Разрешение кнопки "АОсс"
//Coils[1].1;//prm_AObs_Разрешение кнопки "АОбс"
//Coils[1].2;//prm_NOss_Разрешение кнопки "НОсс"
//Coils[1].3;//prm_NObs_Разрешение кнопки "НОбс"
Coils[1].4 := btn.turnUP.prm;//prm_turnUP_Разрешение кнопки "Увеличить обороты"
Coils[1].5 := btn.turnDN.prm;//prm_turnDN_Разрешение кнопки "Уменьшить обороты"
//Coils[1].6;//prm_regNvd_Разрешение кнопки "Регулирование оборотов ВД"
Coils[1].7 := btn.turnUP.prm OR btn.turnDN.prm;//prm_regNst_Разрешение кнопки "Регулирование оборотов СТ"

// ИМы
Coils[4].0		:= am.SK.isON;//NOT dipar_SK_OF_СК открыт
Coils[4].1		:= am.kr1.isON;//dipar_Kr1_ON_Кран КШ1 открыт
Coils[4].2		:= am.Kr1.isOFF;//dipar_Kr1_OF_Кран КШ1 закрыт
Coils[4].3		:= am.Kr2.isON;//dipar_Kr2_ON_Кран КШ2 открыт
Coils[4].4		:= am.Kr2.isOFF;//dipar_Kr2_OF_Кран КШ2 закрыт
Coils[4].5		:= am.Kr4.isON;//dipar_Kr4_ON_Кран КШ4 открыт
Coils[4].6		:= am.Kr4.isOFF;//dipar_Kr4_OF_Кран КШ4 закрыт
Coils[4].7		:= am.Kr5.isON;//dipar_Kr5_ON_Кран КШ5 открыт
Coils[5].0		:= am.Kr5.isOFF;//dipar_Kr5_OF_Кран КШ5 закрыт
Coils[5].1		:= am.Kr6.isON;//dipar_Kr6_ON_Кран КШ6 открыт
Coils[5].2		:= am.Kr6.isOFF;//dipar_Kr6_OF_Кран КШ6 закрыт
Coils[5].3		:= am.Kr9.isON;//dipar_Kr13_ON_Кран КШ13 открыт
Coils[5].4		:= am.Kr9.isOFF;//dipar_Kr13_OF_Кран КШ13 закрыт
Coils[5].5		:= am.Kr12.isON;//dipar_Kr14_ON_Кран КШ14 открыт
Coils[5].6		:= am.Kr12.isOFF;//dipar_Kr14_OF_Кран КШ14 закрыт

// Статусы подсистем
Coils[7].0	:= subsystem.EXT.nrml;	// status_EXT_nrml Внешние сигналы_норма
Coils[7].1	:= subsystem.EXT.alr;	// status_EXT_alr Внешние сигналы_предупрежденеие
Coils[7].2	:= subsystem.EXT.crs;	// status_EXT_crs Внешние сигналы_авария
Coils[7].3	:= subsystem.BD.nrml;	// status_BD_nrml Блок двигателя_норма
Coils[7].4	:= subsystem.BD.alr;	// status_BD_alr Блок двигателя_предупрежденеие
Coils[7].5	:= subsystem.BD.crs;	// status_BD_crs Блок двигателя_авария
Coils[7].6	:= subsystem.MSD.nrml;	// status_MSD_nrml Маслосистема двигателя_норма
Coils[7].7	:= subsystem.MSD.alr;	// status_MSD_alr Маслосистема двигателя_предупрежденеие
Coils[8].0	:= subsystem.MSD.crs;	// status_MSD_crs Маслосистема двигателя_авария
Coils[8].1	:= subsystem.BTG.nrml;	// status_BTG_nrml Блок топливного газа_норма
Coils[8].2	:= subsystem.BTG.alr;	// status_BTG_alr Блок топливного газа_предупрежденеие
Coils[8].3	:= subsystem.BTG.crs;	//status_BTG_crs Блок топливного газа_авария
Coils[8].4	:= subsystem.AVOM.nrml;//status_AVOMD_nrml АВОМД_норма
Coils[8].5	:= subsystem.AVOM.alr;//status_AVOMD_alr АВОМД_предупрежденеие
Coils[8].6	:= subsystem.AVOM.crs;//status_AVOMD_crs АВОМД_авария
Coils[8].7	:= subsystem.BN.nrml;//status_BN_nrml Блок нагнетателя_норма
Coils[9].0	:= subsystem.BN.alr;//status_BN_alr Блок нагнетателя_предупрежденеие
Coils[9].1	:= subsystem.BN.crs;//status_BN_crs Блок нагнетателя_авария
Coils[9].2	:= subsystem.GO.nrml;//status_GO_nrml Газовая обвязка_норма
Coils[9].3	:= subsystem.GO.alr;//status_GO_alr Газовая обвязка_предупрежденеие
Coils[9].4	:= subsystem.GO.crs;//status_GO_crs Газовая обвязка_авария
Coils[9].5	:= subsystem.VS.nrml;//status_VS_nrml Воздушный стартер_норма
Coils[9].6	:= subsystem.VS.alr;//status_VS_alr Воздушный стартер_предупрежденеие
Coils[9].7	:= subsystem.VS.crs;//status_VS_crs Воздушный стартер_авария
Coils[10].0	:= subsystem.BPG.nrml;//status_BPG_nrml Блок пускового газа_норма
Coils[10].1	:= subsystem.BPG.alr;//status_BPG_alr Блок пускового газа_предупрежденеие
Coils[10].2	:= subsystem.BPG.crs;//status_BPG_crs Блок пускового газа_авария
Coils[10].3	:= subsystem.POS.nrml;//status_POS_nrml ПОС ВОУ_норма
Coils[10].4	:= subsystem.POS.alr;//status_POS_alr ПОС ВОУ_предупрежденеие
Coils[10].5	:= subsystem.POS.crs;//status_POS_crs ПОС ВОУ_авария
Coils[10].6	:= subsystem.BU.nrml;//status_BU_nrml Блок автоматики_норма
Coils[10].7	:= subsystem.BU.alr;//status_BU_alr Блок автоматики_предупрежденеие
Coils[11].0	:= subsystem.BU.crs;//status_BU_crs Блок автоматики_авария


// Режим агрегата
General[1]			:= mde.number;

// Аналоги
//Holdings[1]		:= am.APK.pos; 				// aipar_APK_Pos_Положение клапана АПК1		// 2
//StatusReal.0	:= am.APK.flt;
//Holdings[2]		:= 0;			// aipar_reserve									// 4

//Holdings[3]		:= acpar.Ntk.value;		// acpar_evNnd_Расчётная Ntk				// 6
//StatusReal.2	:= acpar.Ntk.flt;

Holdings[4]		:= acpar.Ntk.value;		// acpar_evNvd_Расчётная Ntk				// 8
StatusReal.3	:= acpar.Nst.flt;

Holdings[5]		:= acpar.Nst.value;		// acpar_evNst_Расчётная Nст				// 10
StatusReal.4	:= acpar.Nst.flt;

Holdings[6]		:= aipar.Pg_inN.value;	// acpar_evPg_inN P газа на входе в компрессор		// 12
StatusReal.5	:= aipar.Pg_inN.flt;

Holdings[7]		:= aipar.Pg_outN.value;	// acpar_evPg_outN P газа на выходе из компрессора	// 14
StatusReal.6	:= aipar.Pg_outN.flt;

Holdings[8]		:= aipar.Tg_inN.value;	// acpar_evTg_inN T газа на входе в компрессор		// 16
StatusReal.7	:= aipar.Tg_inN.flt;

Holdings[9]		:= aipar.Tg_outN.value;	// acpar_evTg_outN T газа на выходе из компрессора	// 18
StatusReal.8	:= aipar.Tg_outN.flt;

//Holdings[10]	:= acpar.evdPg_conf.value;	// acpar_evdPg_conf_Расчётная dP газа на аннубар				// 20
//StatusReal.9	:= acpar.evdPg_conf.flt;

Holdings[11]	:= acpar.Tg_inST.value;	// acpar_evTg_outTND_Расчётная Т газа перед СТ					// 22
StatusReal.10	:= acpar.Tg_inST.flt;

//Holdings[12]	:= aipar.Ta_Angar.value;	// acpar_evTa_BN_Расчётная T воздуха в укрытии Компрессора		// 24
//StatusReal.11	:= aipar.Ta_Angar.flt;

Holdings[13]	:= aipar.Ta_inK.value;		// acpar_evTa_inBD_Расчётная T воздуха в блоке двигателя		// 26
StatusReal.12	:= aipar.Ta_inK.flt;

//Holdings[14]	:= s_aspar.surgeRes.value;	// acpar_Surge_Помпажный запас									// 28					
//StatusReal.13	:= s_aspar.surgeRes.flt;

IF aipar.Pg_inN.value > 0.0 THEN
	Holdings[15]	:= aipar.Pg_outN.value / aipar.Pg_inN.value;	// acpar_PR_Степень сжатия // 30
	ELSE 
		Holdings[15] := 0;
END_IF								
StatusReal.14	:= aipar.Pg_outN.flt OR aipar.Pg_inN.flt;		// s_aspar.evPR.flt;

Holdings[16]	:= aipar.Ptg_inTRK.value;	// aipar_Ptg_inD_Р топливного газа на вх. в Д	// 32
StatusReal.15	:= aipar.Ptg_inTRK.flt;

(*
Holdings[1]		:= Holdings[1] + 0.1; 				// aipar_APK_Pos_Положение клапана АПК1		// 2
//Holdings[2]		:= 0;			// aipar_reserve									// 4
Holdings[3]		:= Holdings[3] + 1; 			// acpar_evNnd_Расчётная Nвд							// 6
Holdings[4]		:= 3400;		// acpar_evNvd_Расчётная Nнд				// 8
Holdings[5]		:= 3001;		// acpar_evNst_Расчётная Nст				// 10
Holdings[6]		:= 6.6;	// acpar_evPg_inN_Расчётное P газа на входе в компрессор		// 12
Holdings[7]		:= 7.7;	// acpar_evPg_outN_Расчётное P газа на выходе из компрессора	// 14
Holdings[8]		:= 34.3;	// acpar_evTg_inN_Расчётная T газа на входе в компрессор		// 16
Holdings[9]		:= 87.9;	// acpar_evTg_outN_Расчётная T газа на выходе из компрессора	// 18
Holdings[10]	:= 20.01;	// acpar_evdPg_conf_Расчётная dP газа на аннубар				// 20
Holdings[11]	:= 470;	// acpar_evTg_outTND_Расчётная Т газа перед СТ					// 22
Holdings[12]	:= 22.12;	// acpar_evTa_BN_Расчётная T воздуха в укрытии Компрессора		// 24
Holdings[13]	:= 23.13;		// acpar_evTa_inBD_Расчётная T воздуха в блоке двигателя		// 26
Holdings[14]	:= 67.0;//	acpar. acpar_Surge_Помпажный запас									// 28					
Holdings[15]	:= 0.22;//acpar.PR; acpar_PR_Степень сжатия									// 30
Holdings[16]	:= 19.16;	// aipar_Ptg_inD_Р топливного газа на вх. в Д	// 32
*)
                  
END_PROGRAM

PROGRAM PRG_PRU_TimeSync
VAR
	///  Год, Месяц, День, час, минуты,секунды
	TimeAndDate: ARRAY[0..6] OF WORD;
	UnixTimems: DWORD;
	pres: UDINT;
	pDate: PsTime.SYSTIMEDATE;
END_VAR
VAR CONSTANT
	/// временная зона (в ПРУ Овен отсутствует)
	TimeZone: BYTE := 3;
END_VAR

                    // ---- Синхронизация времени
UnixTimems	:= PsTime.SysTimeRtcGet(pres);
PsTime.SysTimeRtcConvertUtcToDate(UnixTimems, pDate);

TimeAndDate[0]	:= pDate.wYear;				// Год
TimeAndDate[1]	:= pDate.wMonth;			// Месяц
TimeAndDate[2]	:= pDate.wDay;				// День
TimeAndDate[3]	:= pDate.wHour + TimeZone;	// Час
TimeAndDate[4]	:= pDate.wMinute;			// Минуты
TimeAndDate[5]	:= pDate.wSecond;			// Секунды

TimeAndDate[6]	:= 1;		// Признак готовности времени для синхронизации (признак снимается с ПРУ)

// ---- 
                  
END_PROGRAM

FUNCTION ALG_AVOM_Link : BOOL
VAR 
	temperature	: REAL;

END_VAR

                    subsystem.AVOM(
	goWork	:= am.Vn1_AVOM.on OR am.Vn2_AVOM.on OR am.Vn3_AVOM.on OR am.Vn4_AVOM.on,
	goStop	:= NOT ( am.Vn1_AVOM.on OR am.Vn2_AVOM.on OR am.Vn3_AVOM.on OR am.Vn4_AVOM.on ),
	work := am.Vn1_AVOM.isON OR am.Vn2_AVOM.isON OR am.Vn3_AVOM.isON OR am.Vn4_AVOM.isON,
	stop  := NOT ( am.Vn1_AVOM.isON OR am.Vn2_AVOM.isON OR am.Vn3_AVOM.isON OR am.Vn4_AVOM.isON )
);

//enable	:= mde.APK OR alg.work OR alg.NO OR am.PNU.isON OR am.PNS.isON;

avom.AVOM.enable	:= ( avom.AVOM.enable OR fuelreg.fReg.isFire ) AND NOT ( alg.V_000 AND am.PNS.isOFF AND am.PNU.isOFF ); 

temperature := MAX ( aipar.Tm_inD.value, aipar.Tm_outAU.value, aipar.Tm_outAVOM.value );
AVOM.AVOM.update( temperature := temperature );
IF imitGPA.imit_on THEN AVOM_imit(); END_IF;
                  
END_FUNCTION

FUNCTION AVOM_Imit : BOOL
VAR
	temp: REAL;
END_VAR

                    
temp := MAX (aipar.Tm_outD.value, aipar.Ta_inK.value);
aipar.Tm_outAVOM.sim_value	:= aipar.Tm_outAVOM.sim_value + ( temp - ( temp - aipar.Ta_inK.value) * ( TO_BYTE ( am.Vn1_AVOM.isON ) + TO_BYTE ( am.Vn2_AVOM.isON ) + TO_BYTE ( am.Vn3_AVOM.isON ) + TO_BYTE ( am.Vn4_AVOM.isON )) * 0.95 / 4 - aipar.Tm_outAVOM.sim_value ) / tau_Nto0;
aipar.Tm_outAU.sim_value 	:= aipar.Ta_inK.value;
                  
END_FUNCTION

FUNCTION AVOM_Init : BOOL

                    AVOM.AVOM ( Tm_SET		:= tunpar.setTm,
			T1			:= tunpar.T1_avom,
			T2			:= tunpar.T2_avom,
			K			:= tunpar.K_avom,
			DZ			:= tunpar.DZ_avom,
			Vn1_AVOM	:= am.Vn1_AVOM,
			Vn2_AVOM	:= am.Vn2_AVOM,
			Vn3_AVOM	:= am.Vn3_AVOM,
			Vn4_AVOM	:= am.Vn4_AVOM );
                  
END_FUNCTION

FUNCTION ALG_EXT_Link : BOOL

                    subsystem.EXT();
                  
END_FUNCTION

FUNCTION ALG_BTG_Link : BOOL

                    subsystem.BTG();

ALG_BTG_AM();

IF imitGPA.imit_on THEN BTG_imit(); END_IF;
                  
END_FUNCTION

FUNCTION ALG_MSD_link : BOOL

                    subsystem.MSD();

ALG_MSD_AM();

IF imitGPA.imit_on THEN MSD_imit(); END_IF;
                  
END_FUNCTION

FUNCTION MSD_Imit : BOOL
VAR CONSTANT
	dPmg_PNU: REAL := 0.7;
	dpmg_BN: REAL := 2.5;
	Nst_norm: REAL := 8500;
END_VAR

                    
aipar.dPmg.sim_value	:= (aipar.dPmg.value + (dPmg_PNU * BOOL_TO_BYTE( am.PNU.isOn ) + dpmg_BN * acpar.Nst.value / Nst_norm - aipar.dPmg.value) / tau_Po );
                  
END_FUNCTION

FUNCTION ALG_MSD_AM : BOOL

                    tmr.PNU_S_Off.IN 	:= ( NOss.cmd_PNU_S_Off OR AOss.cmd_PNU_S_Off OR Bleeding_full.cmd_PNU_S_Off OR tmr.PNU_S_Off.IN ) AND NOT ( tmr.PNU_S_Off.Q OR tch.Gas_N.value );
tmr.PNU_S_pumpH.IN	:= ( tch.GTDcool.value OR tch.GTDHeat.value ) AND dipar.Pm_N_Pn.value;

am.PNS.on	:= HP.cmd_PNU_S_On OR KPK.cmd_PNU_S_On OR APK.cmd_PNU_S_On OR NOss.cmd_PNU_S_On OR NObs.cmd_PNU_S_On OR AOss.cmd_PNU_S_On OR AObs.cmd_PNU_S_On OR ( mde.GR AND am.PNS.isOFF ) OR tmr.PNU_S_pumpH.IN;
am.PNS.off	:= (( HP.cmd_PNS_Off OR ( mde.HR OR mde.Repair ) AND am.PNS.isON AND tch.nGas_N.value ) AND NOT tmr.PNU_S_Off.IN ) OR Start_D.cmd_PNS_Off OR ( tmr.PNU_S_Off.Q AND tch.nGas_N.value ) OR (( tch.GTDcool.value OR tch.GTDHeat.value OR alg.work ) AND NOT tmr.PNU_S_pumpH.Q AND am.PNS.isON );

am.PNU.on	:= HP.cmd_PNU_S_On OR KPK.cmd_PNU_S_On OR APK.cmd_PNU_S_On OR NOss.cmd_PNU_S_On OR NObs.cmd_PNU_S_On OR AOss.cmd_PNU_S_On OR AObs.cmd_PNU_S_On OR ( mde.GR AND am.PNU.isOFF ) OR tmr.PNU_S_pumpH.IN;
am.PNU.off	:= (( HP.cmd_PNU_Off OR ( mde.HR OR mde.Repair ) AND am.PNU.isON AND tch.nGas_N.value ) AND NOT tmr.PNU_S_Off.IN ) OR Start_D.cmd_PNU_Off OR ( tmr.PNU_S_Off.Q AND tch.nGas_N.value ) OR (( tch.GTDcool.value OR tch.GTDHeat.value OR alg.work ) AND NOT tmr.PNU_S_pumpH.Q AND am.PNU.isON );

// Обогрев маслобака системы смазки
engine.ENBDN( par_value := aipar.Tm_MB.value, par_brk := aipar.Tm_MB.flt, setpoint_value := tunpar.setTmMBDN.value );
engine.ENBDN_HR( par_value := aipar.Tm_MB.value, par_brk := aipar.Tm_MB.flt );
//am.ENBDN.on	:= ( engine.ENBDN_HR.out AND tch.Check_HR.value ) OR engine.ENBDN.out AND NOT ( mde.Repair OR ( mde.HR AND NOT tch.Check_GR.value )) AND alg.reserve; //черепанов добавил alg.reserve

// Обогрев маслобака системы уплотнений
bn.ENBN( par_value := aipar.Tm_MBU.value, par_brk := aipar.Tm_MBU.flt, setpoint_value := tunpar.setTmMBN.value );
bn.ENBN_HR( par_value := aipar.Tm_MBU.value, par_brk := aipar.Tm_MBU.flt );
//am.ENBN.on := ( bn.ENBN_HR.out AND ppu.Check_HR.value ) OR bn.ENBN.out AND NOT ( mde.Repair OR ( mde.HR AND NOT ppu.Check_GR.value )) AND alg.reserve; //черепанов добавил alg.reserve
                  
END_FUNCTION

FUNCTION ALG_BPG_AM : BOOL

                    am.Kr11.on	:= HP.cmd_KR11_On OR Start_D.cmd_KR11_On;
am.Kr11.off	:= HP.cmd_KR11_Off OR Start_D.cmd_KR11_Off OR AOss.cmd_KR11_Off OR AObs.cmd_KR11_Off;

am.Kr10.on	:= am.Kr11.off;
am.Kr10.off	:= am.Kr11.on;

//dopar.Kr10m_ON.value := am.Kr11.on OR am.Kr11.off;
//dopar.Kr11m_ON.value := dopar.Kr11m_ON.value;

                  
END_FUNCTION

FUNCTION ALG_BPG_Link : BOOL

                    subsystem.BPG();

ALG_BPG_AM();

IF imitGPA.imit_on THEN BPG_imit(); END_IF;
                  
END_FUNCTION

FUNCTION BPG_Imit : BOOL

                    
                  
END_FUNCTION

FUNCTION ALG_VS_AM : BOOL

                    am.Kr13.on	:= ( HP.cmd_VS_On OR Start_D.cmd_VS_On OR am.Kr13.on ) AND NOT ( HP.cmd_VS_Off OR Start_D.cmd_VS_Off OR AOss.cmd_VS_Off OR AObs.cmd_VS_Off );
//am.Kr13m.on	:= am.Kr13.on;
                  
END_FUNCTION

FUNCTION ALG_VS_Link : BOOL

                    subsystem.VS(
	goWork	:= am.Kr13.on,
	goStop	:= NOT am.Kr13.on,
	work 	:= am.Kr13.isON,
	stop	:= NOT am.Kr13.isOn
);

ALG_VS_AM();
                  
END_FUNCTION

FUNCTION ALG_BTG_AM : BOOL

                    am.Kr12.on	:= KPK.cmd_KR12_On OR Start_D.cmd_KR12_On;
am.Kr12.off	:= KPK.cmd_KR12_Off OR NOss.cmd_KR12_Off OR NObs.cmd_KR12_Off OR AOss.cmd_KR12_Off OR AObs.cmd_KR12_Off;

am.Kr9.on	:= am.Kr12.off;
am.Kr9.off	:= am.Kr12.on;

//dopar.KR9m_ON.value := am.Kr12.on OR am.Kr12.off;
//dopar.KR12m_ON.value := dopar.KR9m_ON.value;

                  
END_FUNCTION

FUNCTION BTG_Imit : BOOL
VAR CONSTANT
	Ptg: REAL := 2.1;
END_VAR

                    aipar.Ptg_inTRK.sim_value	:= Ptg * BOOL_TO_BYTE ( am.Kr12.isON AND am.Kr9.isOFF );

                  
END_FUNCTION

{region INFO}
(*
 Наименование последовательности: Комплексное тестирование
 Автор: /Разработчик/ 08.08.2025 9:04:03
 Версия: v00.00.18
 Проект: KA107
*)
{endregion}
{attribute 'symbol' := 'none'}
FUNCTION_BLOCK PUBLIC T_testing
VAR_INPUT
	cycle : REAL; //цикл вызова
END_VAR
VAR_OUTPUT
	init : BOOL; //Переинициализирование переменных
	cmd_Nst_5000 : BOOL; //Шаг проверки: Повышение Nст до 5000 об/мин
	finish : BOOL; //Завершение
	{attribute 'symbol' := 'read'}
	drm : Tdrm; //Интерфейсный функциональный блок
END_VAR
VAR
	start : BOOL; //Запуск последовательности
	break : BOOL; //Принудительный выход из последовательности
END_VAR

                    //Собираем переходы для визуализации
drm.transition.0 := start := btn.test_on.out; //Запуск последовательности (0→1): Кнопка "Комплексное тестирование включить"
drm.transition.1 := TRUE; //1→2: Логическая 1
drm.transition.2 := mde.GR; //2→3: Режим ГР
drm.transition.3 := btn.start.prm; //3→4: Разрешение кнопки "Пуск"
drm.transition.4 := HP.finish; //4→5: Последовательность "ХП" завершена
drm.transition.5 := btn.start.prm; //5→6: Разрешение кнопки "Пуск"
drm.transition.6 := KPK.finish; //6→7: Последовательность "КПК" завершена
drm.transition.7 := btn.start.prm; //7→8: Разрешение кнопки "Пуск"
drm.transition.8 := APK.finish; //8→9: Последовательность "АПК" завершена
drm.transition.9 := AOss.finish; //9→10: Последовательность "АОсс" завершена
drm.transition.10 := mde.Repair; //10→11: Режим Ремонт
drm.transition.11 := mde.GR; //11→12: Режим ГР
drm.transition.12 := btn.start.prm; //12→13: Разрешение кнопки "Пуск"
drm.transition.13 := APK.finish; //13→14: Последовательность "АПК" завершена
drm.transition.14 := NOss.finish; //14→15: Последовательность "НОсс" завершена
drm.transition.15 := mde.GR; //15→16: Режим ГР
drm.transition.16 := AObs.finish; //16→17: Последовательность "АОбс" завершена
drm.transition.17 := mde.Repair; //17→18: Режим Ремонт
drm.transition.18 := M_K.finish; //18→19: Последовательность "Переход М-К" завершена
drm.transition.19 := acpar.Nst.value > 4990; //19→20: Nст > 4990 об/мин
drm.transition.20 := K_M.finish; //20→21: Последовательность "Переход К-М" завершена
drm.transition.21 := NObs.finish; //21→22: Последовательность "НОбс" завершена
drm.transition.22 := Bleeding_full.finish; //22→23: Последовательность "Стравливание" завершена
drm.transition.23 := mde.Repair; //23→24: Режим Ремонт
drm.transition.24 := btn.test_off.out; //24→0: Кнопка "Комплексное тестирование отключить"
drm.transition.31 := break := btn.test_off.out; //Принудительный выход из последовательности (N→0): Кнопка "Комплексное тестирование отключить"

//Вызываем экземпляр интерфейсного функционального блока
drm(cycle := cycle);

CASE drm.step OF
-1:	//Сброс команд с предыдущих шагов
	finish := FALSE;
	//Условие запуска последовательности
	//Кнопка "Комплексное тестирование включить"
	IF start AND NOT break THEN drm.step := 1; END_IF;
1:	//Запись уставки таймера шага
	drm.step := 1;//Текущий шаг
	drm.timer_pt := 10; //Таймер: 10 секунд

	//Команды текущего шага
	(*1*) init := drm.cmd.0 := drm.step_time <= cycle; //Переинициализирование переменных

	//Условие перехода (1)→(2)
	//Логическая 1
	IF (TRUE) AND drm.timeout THEN
		drm.cmd := drm.error := 0; drm.timer_pt := cycle; drm.inc := FALSE; drm.step := 2;
		init := FALSE; //Переинициализирование переменных
	END_IF;
2:	//Запись уставки таймера шага
	drm.step := 2;//Текущий шаг
	drm.timer_pt := 10; //Таймер: 10 секунд

	//Команды текущего шага
	(*1*) btn.GR.cmd := drm.cmd.0 := drm.step_time <= cycle; //Шаг проверки: ХП из ГР // Кнопка "ГР"

	//Условие перехода (2)→(3)
	//Режим ГР
	IF (mde.GR) AND drm.timeout THEN
		drm.cmd := drm.error := 0; drm.timer_pt := cycle; drm.inc := FALSE; drm.step := 3;
		btn.GR.cmd := FALSE; //Шаг проверки: ХП из ГР // Кнопка "ГР"
	END_IF;
3:	//Запись уставки таймера шага
	drm.step := 3;//Текущий шаг
	drm.timer_pt := cycle; //Таймер: один цикл вызова

	//Команды текущего шага
	(*1*) btn.HP.cmd := drm.cmd.0 := drm.step_time <= cycle; //Шаг проверки: ХП из ГР // Кнопка "ХП"

	//Условие перехода (3)→(4)
	//Разрешение кнопки "Пуск"
	IF (btn.start.prm) AND drm.timeout THEN
		drm.cmd := drm.error := 0; drm.timer_pt := cycle; drm.inc := FALSE; drm.step := 4;
		btn.HP.cmd := FALSE; //Шаг проверки: ХП из ГР // Кнопка "ХП"
	END_IF;
4:	//Запись уставки таймера шага
	drm.step := 4;//Текущий шаг
	drm.timer_pt := cycle; //Таймер: один цикл вызова

	//Команды текущего шага
	(*1*) btn.Start.cmd := drm.cmd.0 := drm.step_time <= cycle; //Шаг проверки: ХП из ГР // Кнопка "Пуск"

	//Условие перехода (4)→(5)
	//Последовательность "ХП" завершена
	IF (HP.finish) AND drm.timeout THEN
		drm.cmd := drm.error := 0; drm.timer_pt := cycle; drm.inc := FALSE; drm.step := 5;
		btn.Start.cmd := FALSE; //Шаг проверки: ХП из ГР // Кнопка "Пуск"
	END_IF;
5:	//Запись уставки таймера шага
	drm.step := 5;//Текущий шаг
	drm.timer_pt := cycle; //Таймер: один цикл вызова

	//Команды текущего шага
	(*1*) btn.KPK.cmd := drm.cmd.0 := drm.step_time <= cycle; //Шаг проверки: КПК из ГР // Кнопка "КПК"

	//Условие перехода (5)→(6)
	//Разрешение кнопки "Пуск"
	IF (btn.start.prm) AND drm.timeout THEN
		drm.cmd := drm.error := 0; drm.timer_pt := cycle; drm.inc := FALSE; drm.step := 6;
		btn.KPK.cmd := FALSE; //Шаг проверки: КПК из ГР // Кнопка "КПК"
	END_IF;
6:	//Запись уставки таймера шага
	drm.step := 6;//Текущий шаг
	drm.timer_pt := cycle; //Таймер: один цикл вызова

	//Команды текущего шага
	(*1*) btn.Start.cmd := drm.cmd.0 := drm.step_time <= cycle; //Шаг проверки: КПК из ГР // Кнопка "Пуск"

	//Условие перехода (6)→(7)
	//Последовательность "КПК" завершена
	IF (KPK.finish) AND drm.timeout THEN
		drm.cmd := drm.error := 0; drm.timer_pt := cycle; drm.inc := FALSE; drm.step := 7;
		btn.Start.cmd := FALSE; //Шаг проверки: КПК из ГР // Кнопка "Пуск"
	END_IF;
7:	//Запись уставки таймера шага
	drm.step := 7;//Текущий шаг
	drm.timer_pt := cycle; //Таймер: один цикл вызова

	//Команды текущего шага
	(*1*) btn.APK.cmd := drm.cmd.0 := drm.step_time <= cycle; //Шаг проверки: АПК из ГР под газом // Кнопка "АПК"

	//Условие перехода (7)→(8)
	//Разрешение кнопки "Пуск"
	IF (btn.start.prm) AND drm.timeout THEN
		drm.cmd := drm.error := 0; drm.timer_pt := cycle; drm.inc := FALSE; drm.step := 8;
		btn.APK.cmd := FALSE; //Шаг проверки: АПК из ГР под газом // Кнопка "АПК"
	END_IF;
8:	//Запись уставки таймера шага
	drm.step := 8;//Текущий шаг
	drm.timer_pt := cycle; //Таймер: один цикл вызова

	//Команды текущего шага
	(*1*) btn.Start.cmd := drm.cmd.0 := drm.step_time <= cycle; //Шаг проверки: АПК из ГР под газом // Кнопка "Пуск"

	//Условие перехода (8)→(9)
	//Последовательность "АПК" завершена
	IF (APK.finish) AND drm.timeout THEN
		drm.cmd := drm.error := 0; drm.timer_pt := cycle; drm.inc := FALSE; drm.step := 9;
		btn.Start.cmd := FALSE; //Шаг проверки: АПК из ГР под газом // Кнопка "Пуск"
	END_IF;
9:	//Запись уставки таймера шага
	drm.step := 9;//Текущий шаг
	drm.timer_pt := cycle; //Таймер: один цикл вызова

	//Команды текущего шага
	(*1*) btn.AOss.cmd := drm.cmd.0 := drm.step_time <= cycle; //Шаг проверки: АОсс из Кольца // Кнопка "АОсс"

	//Условие перехода (9)→(10)
	//Последовательность "АОсс" завершена
	IF (AOss.finish) AND drm.timeout THEN
		drm.cmd := drm.error := 0; drm.timer_pt := cycle; drm.inc := FALSE; drm.step := 10;
		btn.AOss.cmd := FALSE; //Шаг проверки: АОсс из Кольца // Кнопка "АОсс"
	END_IF;
10:	//Запись уставки таймера шага
	drm.step := 10;//Текущий шаг
	drm.timer_pt := 10; //Таймер: 10 секунд

	//Команды текущего шага
	(*1*) btn.Unlock.cmd := drm.cmd.0 := drm.step_time <= cycle; //Шаг проверки: АОсс из Кольца // Кнопка "Деблокировка"

	//Условие перехода (10)→(11)
	//Режим Ремонт
	IF (mde.Repair) AND drm.timeout THEN
		drm.cmd := drm.error := 0; drm.timer_pt := cycle; drm.inc := FALSE; drm.step := 11;
		btn.Unlock.cmd := FALSE; //Шаг проверки: АОсс из Кольца // Кнопка "Деблокировка"
	END_IF;
11:	//Запись уставки таймера шага
	drm.step := 11;//Текущий шаг
	drm.timer_pt := 10; //Таймер: 10 секунд

	//Команды текущего шага
	(*1*) btn.GR.cmd := drm.cmd.0 := drm.step_time <= cycle; //Шаг проверки: АПК из ГР без газа // Кнопка "ГР"

	//Условие перехода (11)→(12)
	//Режим ГР
	IF (mde.GR) AND drm.timeout THEN
		drm.cmd := drm.error := 0; drm.timer_pt := cycle; drm.inc := FALSE; drm.step := 12;
		btn.GR.cmd := FALSE; //Шаг проверки: АПК из ГР без газа // Кнопка "ГР"
	END_IF;
12:	//Запись уставки таймера шага
	drm.step := 12;//Текущий шаг
	drm.timer_pt := cycle; //Таймер: один цикл вызова

	//Команды текущего шага
	(*1*) btn.APK.cmd := drm.cmd.0 := drm.step_time <= cycle; //Шаг проверки: АПК из ГР без газа // Кнопка "АПК"

	//Условие перехода (12)→(13)
	//Разрешение кнопки "Пуск"
	IF (btn.start.prm) AND drm.timeout THEN
		drm.cmd := drm.error := 0; drm.timer_pt := cycle; drm.inc := FALSE; drm.step := 13;
		btn.APK.cmd := FALSE; //Шаг проверки: АПК из ГР без газа // Кнопка "АПК"
	END_IF;
13:	//Запись уставки таймера шага
	drm.step := 13;//Текущий шаг
	drm.timer_pt := cycle; //Таймер: один цикл вызова

	//Команды текущего шага
	(*1*) btn.Start.cmd := drm.cmd.0 := drm.step_time <= cycle; //Шаг проверки: АПК из ГР без газа // Кнопка "Пуск"

	//Условие перехода (13)→(14)
	//Последовательность "АПК" завершена
	IF (APK.finish) AND drm.timeout THEN
		drm.cmd := drm.error := 0; drm.timer_pt := cycle; drm.inc := FALSE; drm.step := 14;
		btn.Start.cmd := FALSE; //Шаг проверки: АПК из ГР без газа // Кнопка "Пуск"
	END_IF;
14:	//Запись уставки таймера шага
	drm.step := 14;//Текущий шаг
	drm.timer_pt := cycle; //Таймер: один цикл вызова

	//Команды текущего шага
	(*1*) btn.NOss.cmd := drm.cmd.0 := drm.step_time <= cycle; //Шаг проверки: НОсс из Кольца // Кнопка "НОсс"

	//Условие перехода (14)→(15)
	//Последовательность "НОсс" завершена
	IF (NOss.finish) AND drm.timeout THEN
		drm.cmd := drm.error := 0; drm.timer_pt := cycle; drm.inc := FALSE; drm.step := 15;
		btn.NOss.cmd := FALSE; //Шаг проверки: НОсс из Кольца // Кнопка "НОсс"
	END_IF;
15:	//Запись уставки таймера шага
	drm.step := 15;//Текущий шаг
	drm.timer_pt := 10; //Таймер: 10 секунд

	//Команды текущего шага
	(*1*) btn.GR.cmd := drm.cmd.0 := drm.step_time <= cycle; //Шаг проверки: АПМ из ГР без газа // Кнопка "ГР"

	//Условие перехода (15)→(16)
	//Режим ГР
	IF (mde.GR) AND drm.timeout THEN
		drm.cmd := drm.error := 0; drm.timer_pt := cycle; drm.inc := FALSE; drm.step := 16;
		btn.GR.cmd := FALSE; //Шаг проверки: АПМ из ГР без газа // Кнопка "ГР"
	END_IF;
16:	//Запись уставки таймера шага
	drm.step := 16;//Текущий шаг
	drm.timer_pt := cycle; //Таймер: один цикл вызова

	//Команды текущего шага
	(*1*) btn.AObs.cmd := drm.cmd.0 := drm.step_time <= cycle; //Шаг проверки: АОбс из Магистрали // Кнопка "АОбс"

	//Условие перехода (16)→(17)
	//Последовательность "АОбс" завершена
	IF (AObs.finish) AND drm.timeout THEN
		drm.cmd := drm.error := 0; drm.timer_pt := cycle; drm.inc := FALSE; drm.step := 17;
		btn.AObs.cmd := FALSE; //Шаг проверки: АОбс из Магистрали // Кнопка "АОбс"
	END_IF;
17:	//Запись уставки таймера шага
	drm.step := 17;//Текущий шаг
	drm.timer_pt := 10; //Таймер: 10 секунд

	//Команды текущего шага
	(*1*) btn.Unlock.cmd := drm.cmd.0 := drm.step_time <= cycle; //Шаг проверки: АОбс из Магистрали // Кнопка "Деблокировка"

	//Условие перехода (17)→(18)
	//Режим Ремонт
	IF (mde.Repair) AND drm.timeout THEN
		drm.cmd := drm.error := 0; drm.timer_pt := cycle; drm.inc := FALSE; drm.step := 18;
		btn.Unlock.cmd := FALSE; //Шаг проверки: АОбс из Магистрали // Кнопка "Деблокировка"
	END_IF;
18:	//Запись уставки таймера шага
	drm.step := 18;//Текущий шаг
	drm.timer_pt := cycle; //Таймер: один цикл вызова

	//Команды текущего шага
	(*1*) btn.M_K.cmd := drm.cmd.0 := drm.step_time <= cycle; //Шаг проверки: Переход М-К // Кнопка "Переход М-К"

	//Условие перехода (18)→(19)
	//Последовательность "Переход М-К" завершена
	IF (M_K.finish) AND drm.timeout THEN
		drm.cmd := drm.error := 0; drm.timer_pt := cycle; drm.inc := FALSE; drm.step := 19;
		btn.M_K.cmd := FALSE; //Шаг проверки: Переход М-К // Кнопка "Переход М-К"
	END_IF;
19:	//Запись уставки таймера шага
	drm.step := 19;//Текущий шаг
	drm.timer_pt := cycle; //Таймер: один цикл вызова

	//Команды текущего шага
	(*1*) cmd_Nst_5000 := drm.cmd.0 := drm.step_time <= cycle; //Шаг проверки: Повышение Nст до 5000 об/мин
	(*1*) drm.error.0 := acpar.Nst.value < 5000; //Nст < 5000 об/мин

	//Условие перехода (19)→(20)
	//Nст > 4990 об/мин
	IF (acpar.Nst.value > 4990) AND drm.timeout THEN
		drm.cmd := drm.error := 0; drm.timer_pt := cycle; drm.inc := FALSE; drm.step := 20;
		cmd_Nst_5000 := FALSE; //Шаг проверки: Повышение Nст до 5000 об/мин
	END_IF;
20:	//Запись уставки таймера шага
	drm.step := 20;//Текущий шаг
	drm.timer_pt := cycle; //Таймер: один цикл вызова

	//Команды текущего шага
	(*1*) btn.K_M.cmd := drm.cmd.0 := drm.step_time <= cycle; //Шаг проверки: Переход К-М // Кнопка "Переход К-М"

